// TwinCAT 3 PLC project MiseEnRoute
// libraries:
//   Maxon,1.0.0.0,Maxon Motor
//   Tc2_Standard,newest,Beckhoff Automation GmbH
//   Tc2_System,newest,Beckhoff Automation GmbH
//   Tc2_Utilities,newest,Beckhoff Automation GmbH
//   Tc3_Interfaces,3.3.0.0,Beckhoff Automation GmbH
//   Tc3_Module,3.3.6.0,Beckhoff Automation GmbH
// project tree:
//   / Blinking.TcTTO, GlobalImagePool.TcIPO (not stored), GlobalTextList.TcGTLO, Slow_Tasks.TcTTO, Standard.TcTTO, TestOperator.TcTTO, Visualization Manager.TcVMO (not stored)
//   Data types/ ETHERCAT.TcDUT, FLAGS.TcDUT, FLOWMETER_CONTROL.TcDUT, FLOWMETER_SENSOR.TcDUT, FLOWMETER_VALUES.TcDUT, GEN_PARAMS.TcDUT, HMI_DB_ADS.TcDUT, PANEL_KEYS.TcDUT, PANEL_LEDS.TcDUT, PMAX_DI.TcDUT, PMAX_DO.TcDUT, POW_DI.TcDUT, POW_DO.TcDUT, PRESSURE_SENSOR.TcDUT, PRINT_DI.TcDUT, PRINT_DO.TcDUT, PROG_STEPS.TcDUT, PUMP_PARAMS.TcDUT, PUMP_PARAMS_DB.TcDUT, Q_DI.TcDUT, Q_DO.TcDUT, SAFETY_IN.TcDUT, SAFETY_OUT.TcDUT, VAC_DI.TcDUT, VAC_DO.TcDUT
//   Global Variables/ Constant_Variables.TcGVL, Events_Variables.TcGVL, Flag_Variables.TcGVL, IOs_Variables.TcGVL, TwinCAT_Configuration.TcGVL, Variable_Configuration.TcGVL
//   POUs/ AIS.TcPOU, CHECK_VALVES_SENSORS.TcPOU, EVENTS.TcPOU, GEMMA.TcPOU, MAIN.TcPOU, Q1_MOTOR.TcPOU, Q2_MOTOR.TcPOU, SAFETY.TcPOU, testop.TcPOU, USB.TcPOU
//   POUs/Carriers/ CONVEYOR.TcPOU, JIG.TcPOU, JIG_2ND.TcPOU
//   POUs/EH/ EH_FLOMETER.TcPOU, EH_IEEE754_TO_REAL.TcPOU
//   POUs/Functions/ CONVERT_MASS_TO_FLOW.TcPOU
//   POUs/HMI/ LEDS.TcPOU
//   POUs/Stations/ PMAX.TcPOU, PRINT.TcPOU, Q1.TcPOU, Q2.TcPOU, VAC.TcPOU
//   POUs/Water/ WATER_TANK.TcPOU, WATER_TANKS.TcPOU
//   POUs/WIKA/ WIKA_GET_VALUES.TcPOU
//   Visualizations/ FLAGS.TcVIS, GEMMA.TcVIS, Motor.TcVIS, P_MAX.TcVIS, Q1.TcVIS, Q2.TcVIS, VAC.TcVIS

CONFIGURATION MiseEnRoute
    RESOURCE PLC ON TwinCAT3
        TASK Blinking(INTERVAL := T#450000us, PRIORITY := 23);
        TASK Slow_Tasks(INTERVAL := T#200000us, PRIORITY := 22);
        TASK Standard(INTERVAL := T#10ms, PRIORITY := 20);
        TASK TestOperator(INTERVAL := T#100000us, PRIORITY := 21);
        PROGRAM LEDS WITH Blinking : LEDS;
        PROGRAM USB WITH Slow_Tasks : USB;
        PROGRAM MAIN WITH Standard : MAIN;
        PROGRAM testop WITH TestOperator : testop;
    END_RESOURCE
END_CONFIGURATION

// ---- Data types/ETHERCAT.TcDUT
TYPE ETHERCAT :
STRUCT

	POW_COUPLER_STATUS:UINT;
	VAC_COUPLER_STATUS:UINT;
	Q1_COUPLER_STATUS:UINT;
	Q2_COUPLER_STATUS:UINT;
	PMAX_COUPLER_STATUS:UINT;
	PRINT_COUPLER_STATUS:UINT;

END_STRUCT
END_TYPE

// ---- Data types/FLAGS.TcDUT
TYPE FLAGS :
STRUCT

	INIT_OK:BOOL;
	INIT_CHECK_VALVES_SENSORS:BOOL;
	SAFETY_OK:BOOL;
	MANUAL:BOOL;
	AUTO:BOOL;
	VAC_STATUS: BOOL;
	JIG_VAC_STATUS: BOOL;
	Q1_STATUS: BOOL;
	Q2_STATUS: BOOL;
	PMAX_STATUS: BOOL;
	PRINT_STATUS: BOOL;
	JIG_Q1_STATUS: BOOL;
	JIG_Q2_STATUS: BOOL;
	JIG_PMAX_STATUS: BOOL;
	JIG_PRINT_STATUS: BOOL;
	VAC_RELEASE_CARRIER:BOOL;
	Q1_RELEASE_CARRIER:BOOL;
	Q2_RELEASE_CARRIER:BOOL;
	PMAX_RELEASE_CARRIER:BOOL;
	PRINT_RELEASE_CARRIER:BOOL;
	DOORS_OPEN:BOOL;
	F2_END:BOOL;
	GEMMA: STRING;
	MOTOR_Q1_INIT_OK:BOOL;
	MOTOR_Q1_POSITION:DINT;
	MOTOR_Q2_INIT_OK:BOOL;
	MOTOR_Q2_POSITION:DINT;



END_STRUCT
END_TYPE

// ---- Data types/FLOWMETER_CONTROL.TcDUT
TYPE FLOWMETER_CONTROL :
STRUCT

	SET_TOT: USINT;
	SET_MODE: USINT;

END_STRUCT
END_TYPE

// ---- Data types/FLOWMETER_SENSOR.TcDUT

(************************************************************************************************
*
*Variables structure for E&H flowmeter PROMAS 83A
*
***********************************************************************************************)


TYPE FLOWMETER_SENSOR :
STRUCT

	A1 :ARRAY[0..4] OF USINT;
	A2 :ARRAY[0..4] OF USINT;
	A3 :ARRAY[0..4] OF USINT;
	A4 :ARRAY[0..4] OF USINT;
	A5 :ARRAY[0..4] OF USINT;
	A6 :ARRAY[0..4] OF USINT;
	TOT :ARRAY[0..4] OF USINT;

END_STRUCT
END_TYPE

// ---- Data types/FLOWMETER_VALUES.TcDUT
TYPE FLOWMETER_VALUES :
STRUCT
	MassFlow:REAL;
	VolumeFlow:REAL;
	CorrectedVolueFLow:REAL;
	Density:REAL;
	ReferenceDensity:REAL;
	Temperature:REAL;
	TotalMass:REAL;
END_STRUCT
END_TYPE

// ---- Data types/GEN_PARAMS.TcDUT
TYPE GEN_PARAMS :
STRUCT

	USE_JIG_OP2:BOOL:=TRUE; (*Use or not the jig for the operator 2 - Right - *)

END_STRUCT
	END_TYPE

// ---- Data types/HMI_DB_ADS.TcDUT
TYPE HMI_DB_ADS :
STRUCT

	MANUAL				:REAL; (*Variables en provenance de la DB depuis le HMI*)
	AUTO				:REAL;
	NOT_AUS_RESET		:REAL;


END_STRUCT
END_TYPE

// ---- Data types/PANEL_KEYS.TcDUT
TYPE PANEL_KEYS :
STRUCT

	KEY1:BOOL;
	KEY2:BOOL;
	KEY3:BOOL;
	KEY4:BOOL;
	KEY5:BOOL;
	KEY6:BOOL;
	KEY7:BOOL;
	KEY8:BOOL;
	KEY9:BOOL;
	KEY10:BOOL;


END_STRUCT
END_TYPE

// ---- Data types/PANEL_LEDS.TcDUT
TYPE PANEL_LEDS :
STRUCT

	LED1:BOOL;
	LED2:BOOL;
	LED3:BOOL;
	LED4:BOOL;
	LED5:BOOL;
	LED6:BOOL;
	LED7:BOOL;
	LED8:BOOL;
	LED9:BOOL;
	LED10:BOOL;


END_STRUCT
END_TYPE

// ---- Data types/PMAX_DI.TcDUT
(************************************************************************************************
*
*Max pressure DI
*
***********************************************************************************************)

TYPE PMAX_DI :
STRUCT

	WAGON_WAITING:BOOL;
	WAGON_PRESENT:BOOL;
	WAGON_AWAY:BOOL;
	CYLINDER_TOP_IN:BOOL;
	CYLINDER_TOP_OUT:BOOL;
	CYLINDER_BOT_IN:BOOL;
	CYLINDER_BOT_OUT:BOOL;
	POWER_CYLINDER_IN:BOOL;
	POWER_CYLINDER_OUT:BOOL;
	Q3_OK:BOOL; 					(*Alim pompe*)
	WATER_TANK_HIGH:BOOL;
	WATER_TANK_LOW:BOOL;

END_STRUCT
END_TYPE

// ---- Data types/PMAX_DO.TcDUT
(************************************************************************************************
*
*Max pressure DO
*
***********************************************************************************************)

TYPE PMAX_DO :
STRUCT

	WAGON_WAIT_CYLINDER:BOOL;
	WAGON_LOCK_CYLINDER:BOOL;
	WAGON_STOP_CYLINDER:BOOL;
	HYDRO_CYLINDER_TOP:BOOL;
	HYDRO_CYLINDER_BOT:BOOL;
	ELECTR_CYLINDER:BOOL;
	Y7:BOOL;
	Y8:BOOL;
	PUMP_POWER:BOOL;
	PRESSURE_VALVE:BOOL;
	WATER_TANK_VALVE:BOOL;
	FLOW_STOP_VALVE:BOOL;
	FLOW_STOP_BOTT:BOOL;

END_STRUCT
END_TYPE

// ---- Data types/POW_DI.TcDUT

(************************************************************************************************
*
*Variables structure for the digitals intputs of the POWER module
*
***********************************************************************************************)


TYPE POW_DI :
STRUCT

	Q5_OK:BOOL; 		(* Disjoncteur Alimentation Chroma OK*)
	Q6_OK:BOOL;		(* Disjoncteur Alimentation Stations OK*)
	Q7_OK:BOOL;			(* Disjoncteur Moteurs L1L2L3 OK*)
	Q8_OK:BOOL;		(* Protection moteur 1 OK *)
	Q9_OK:BOOL;		(* Protection moteur 2 OK*)
	Q10_OK:BOOL;		(* Protection moteur 3 OK*)
	Q11_OK:BOOL;		(* Protection moteur 4 OK*)

END_STRUCT
END_TYPE

// ---- Data types/POW_DO.TcDUT

(************************************************************************************************
*
*Variables structure for the digitals ouputs of the POWER module
*
***********************************************************************************************)

TYPE POW_DO :
STRUCT

	HMI_LED_GREEN:BOOL;
	HMI_LED_ORANGE:BOOL;
	HMI_LED_RED:BOOL;
	HMI_LED_BLUE:BOOL;
	CONVEYOR_RELAIS:BOOL;


END_STRUCT
END_TYPE

// ---- Data types/PRESSURE_SENSOR.TcDUT

(************************************************************************************************
*
*Variables structure for WIKA pressure sensor
*
***********************************************************************************************)

TYPE PRESSURE_SENSOR :
STRUCT

	VALUE :ARRAY [0..7] OF USINT;

END_STRUCT
END_TYPE

// ---- Data types/PRINT_DI.TcDUT
(************************************************************************************************
*
*Printer DI
*
***********************************************************************************************)


TYPE PRINT_DI :
STRUCT

	WAGON_WAITING:BOOL;
	WAGON_PRESENT:BOOL;
	WAGON_AWAY:BOOL;
	Q3_OK:BOOL; 					(*Alim pompe*)
	WATER_TANK_HIGH:BOOL;
	WATER_TANK_LOW:BOOL;
	ASK_RELEASE_JIG_OP1:BOOL;
	ASK_RELEASE_JIG_OP2:BOOL;
	GRIPPER_OPEN:BOOL;
	GRIPPER_CLOSED:BOOL;
	X_IN:BOOL;
	X_OUT:BOOL;
	Z_UP:BOOL;
	Z_DOWN:BOOL;

END_STRUCT
END_TYPE

// ---- Data types/PRINT_DO.TcDUT
(************************************************************************************************
*
*Printer DO
*
***********************************************************************************************)

TYPE PRINT_DO :
STRUCT

	WAGON_WAIT_CYLINDER:BOOL;
	WAGON_LOCK_CYLINDER:BOOL;
	WAGON_STOP_CYLINDER:BOOL;
	EJECTION_CYLINDER_X:BOOL;
	EJECTION_CYLINDER_Z:BOOL;
	EJECTION_GRIPPER:BOOL;
	Y7:BOOL;
	Y8:BOOL;
	PUMP_POWER:BOOL;
	WATER_TANK_VALVE:BOOL;

END_STRUCT
END_TYPE

// ---- Data types/PROG_STEPS.TcDUT
TYPE PROG_STEPS :
STRUCT

	VAC_STEP:INT;
	Q1_STEP:INT;
	Q2_STEP:INT;
	PMAX_STEP:INT;
	PRINT_STEP:INT;


END_STRUCT
END_TYPE

// ---- Data types/PUMP_PARAMS.TcDUT
TYPE PUMP_PARAMS :
STRUCT

	VAC_ENABLE:BOOL					:=FALSE;				(*Enable Test*)
	VAC_PUMPING_TIME:TIME			:=T#5s; 			(*Pumping delay to prepare the pump for the suction test *)
	VAC_MEASUREMENT_TIME:TIME		:=T#5s; 			(*Measurement time for the sunction pressure *)
	VAC_PRESSURE_LIMIT:REAL			:=-0.7; 			(*Vacuum pressure Limit Higher than this parameter -> NO GOOD [bar]*)

	Q1_ENABLE:BOOL					:=TRUE;				(*Enable Test*)
	Q1_PUMPING_TIME:TIME			:=T#20s; 			(*Pumping delay to prepare the pump for the flow rate test *)
	Q1_MEASUREMENT_TIME:TIME		:=T#10s; 			(*Measurement time for the flow rate*)
	Q1_FLOW_TARGET:REAL				:=350; 				(*Flow rate target [ml/min]*)
	Q1_FLOW_LIMIT_UP:REAL			:=800; 				(*Flow rate Uper limit. Q>This limit -> NO GOOD [ml/min]*)
	Q1_FLOW_LIMIT_DOWN:REAL			:=100; 				(*Flow rate Lower limit. Q<This limit -> NO GOOD [ml/min]*)
	Q1_PRESSURE_TARGET:REAL			:=8; 				(*Pressure target [bar]*)
	Q1_PRESSURE_LIMIT_UP:REAL		:=15; 				(*Pressure Uper limit. p>This limit -> NO GOOD [bar]*)
	Q1_PRESSURE_LIMIT_DOWN:REAL		:=4;	 			(*Pressure Lower limit. p<This limit -> NO GOOD [bar]*)
	Q1_MAX_FLOW:BOOL				:=FALSE;			(*Use the max flow bypass*)

	Q2_ENABLE:BOOL					:=TRUE;				(*Enable Test*)
	Q2_PUMPING_TIME:TIME			:=T#20s; 			(*Pumping delay to prepare the pump for the flow rate test *)
	Q2_MEASUREMENT_TIME:TIME		:=T#10s; 			(*Measurement time for the flow rate*)
	Q2_FLOW_TARGET:REAL				:=350; 				(*Flow rate target [ml/min]*)
	Q2_FLOW_LIMIT_UP:REAL			:=800; 				(*Flow rate Uper limit. Q>This limit -> NO GOOD [ml/min]*)
	Q2_FLOW_LIMIT_DOWN:REAL			:=100; 				(*Flow rate Lower limit. Q<This limit -> NO GOOD [ml/min]*)
	Q2_PRESSURE_TARGET:REAL			:=8; 				(*Pressure target [bar]*)
	Q2_PRESSURE_LIMIT_UP:REAL		:=15; 				(*Pressure Uper limit. p>This limit -> NO GOOD [bar]*)
	Q2_PRESSURE_LIMIT_DOWN:REAL		:=4;	 			(*Pressure Lower limit. p<This limit -> NO GOOD [bar]*)
	Q2_MAX_FLOW:BOOL				:=FALSE;			(*Use the max flow bypass*)

	PMAX_ENABLE:BOOL				:=FALSE;				(*Enable Test*)
	PMAX_PUMPING_TIME:TIME			:=T#10s; 			(*Pumping delay to prepare the pump for the max pressure test *)
	PMAX_MEASUREMENT_TIME:TIME		:=T#8s; 			(*Measurement time for the max pressure test *)
	PMAX_PRESSURE_LIMIT:REAL		:=10; 				(*Max pressure lower than this parameter -> NO GOOD [bar]*)
	PMAX_PRESSURE_LOOSE_TIME:TIME	:=T#3s;				(*Valves Tightness test duration*)

	PRINT_ENABLE:BOOL				:=TRUE;			(*Enable Test*)

END_STRUCT
END_TYPE

// ---- Data types/PUMP_PARAMS_DB.TcDUT
TYPE PUMP_PARAMS_DB :
STRUCT


	VAC_ENABLE:REAL					;				(*Enable Test*)
	VAC_PUMPING_TIME:REAL			; 				(*Pumping delay to prepare the pump for the suction test *)
	VAC_MEASUREMENT_TIME:REAL		; 				(*Measurement time for the sunction pressure *)
	VAC_PRESSURE_LIMIT:REAL			; 				(*Vacuum pressure Limit Higher than this parameter -> NO GOOD [bar]*)

	Q1_ENABLE:REAL					;				(*Enable Test*)
	Q1_PUMPING_TIME:REAL				; 				(*Pumping delay to prepare the pump for the flow rate test *)
	Q1_MEASUREMENT_TIME:REAL		; 				(*Measurement time for the flow rate*)
	Q1_FLOW_TARGET:REAL				; 				(*Flow rate target [ml/min]*)
	Q1_FLOW_LIMIT_UP:REAL				; 				(*Flow rate Uper limit. Q>This limit -> NO GOOD [ml/min]*)
	Q1_FLOW_LIMIT_DOWN:REAL			; 				(*Flow rate Lower limit. Q<This limit -> NO GOOD [ml/min]*)
	Q1_PRESSURE_TARGET:REAL		; 				(*Pressure target [bar]*)
	Q1_PRESSURE_LIMIT_UP:REAL		; 				(*Pressure Uper limit. p>This limit -> NO GOOD [bar]*)
	Q1_PRESSURE_LIMIT_DOWN:REAL	;	 			(*Pressure Lower limit. p<This limit -> NO GOOD [bar]*)
	Q1_MAX_FLOW:REAL					;				(*Use the max flow bypass*)

	Q2_ENABLE:REAL					;				(*Enable Test*)
	Q2_PUMPING_TIME:REAL				; 				(*Pumping delay to prepare the pump for the flow rate test *)
	Q2_MEASUREMENT_TIME:REAL		; 				(*Measurement time for the flow rate*)
	Q2_FLOW_TARGET:REAL				; 				(*Flow rate target [ml/min]*)
	Q2_FLOW_LIMIT_UP:REAL				; 				(*Flow rate Uper limit. Q>This limit -> NO GOOD [ml/min]*)
	Q2_FLOW_LIMIT_DOWN:REAL			; 				(*Flow rate Lower limit. Q<This limit -> NO GOOD [ml/min]*)
	Q2_PRESSURE_TARGET:REAL		; 				(*Pressure target [bar]*)
	Q2_PRESSURE_LIMIT_UP:REAL		; 				(*Pressure Uper limit. p>This limit -> NO GOOD [bar]*)
	Q2_PRESSURE_LIMIT_DOWN:REAL	;	 			(*Pressure Lower limit. p<This limit -> NO GOOD [bar]*)
	Q2_MAX_FLOW:REAL					;				(*Use the max flow bypass*)

	PMAX_ENABLE:REAL					;				(*Enable Test*)
	PMAX_PUMPING_TIME:REAL			; 				(*Pumping delay to prepare the pump for the max pressure test *)
	PMAX_MEASUREMENT_TIME:REAL	; 				(*Measurement time for the max pressure test *)
	PMAX_PRESSURE_LIMIT:REAL		; 				(*Max pressure lower than this parameter -> NO GOOD [bar]*)

	PRINT_ENABLE:REAL				;				(*Enable Test*)


END_STRUCT
END_TYPE

// ---- Data types/Q_DI.TcDUT
(************************************************************************************************
*
*Flowmeter stations DI
*
***********************************************************************************************)

TYPE Q_DI :
STRUCT


	WAGON_WAITING:BOOL;
	WAGON_PRESENT:BOOL;
	WAGON_AWAY:BOOL;
	CYLINDER_TOP_IN:BOOL;
	CYLINDER_TOP_OUT:BOOL;
	CYLINDER_BOT_IN:BOOL;
	CYLINDER_BOT_OUT:BOOL;
	POWER_CYLINDER_IN:BOOL;
	POWER_CYLINDER_OUT:BOOL;
	Q3_OK:BOOL; 					(*Alim pompe*)
	WATER_TANK_HIGH:BOOL;
	WATER_TANK_LOW:BOOL;

END_STRUCT
END_TYPE

// ---- Data types/Q_DO.TcDUT
(************************************************************************************************
*
*Flowmeter stations DI
*
***********************************************************************************************)

TYPE Q_DO :
STRUCT


	WAGON_WAIT_CYLINDER:BOOL;
	WAGON_LOCK_CYLINDER:BOOL;
	WAGON_STOP_CYLINDER:BOOL;
	HYDRO_CYLINDER_TOP:BOOL;
	HYDRO_CYLINDER_BOT:BOOL;
	ELECTR_CYLINDER:BOOL;
	Y7:BOOL;
	Y8:BOOL;
	PUMP_POWER:BOOL;
	MAX_FLOW_VALVE:BOOL;
	WATER_TANK_VALVE:BOOL;
	FLOW_STOP_VALVE:BOOL;
	FLOW_STOP_BOTT:BOOL;

END_STRUCT
END_TYPE

// ---- Data types/SAFETY_IN.TcDUT
TYPE SAFETY_IN :
STRUCT

	DOORS_FBerr:BOOL;
	DOORS_COMerr:BOOL;
	DOORS_State:USINT;
	DOOR_VAC_CLOSED:BOOL;
	DOOR_Q1_CLOSED:BOOL;
	DOOR_Q2_CLOSED:BOOL;
	DOOR_PMAX_CLOSED:BOOL;
	DOOR_PRINT_CLOSED:BOOL;

	NOT_AUS_FBerr:BOOL;
	NOT_AUS_COMerr:BOOL;
	NOT_AUS_State:USINT;

END_STRUCT
END_TYPE

// ---- Data types/SAFETY_OUT.TcDUT
TYPE SAFETY_OUT :
STRUCT

	DOORS_RUN:BOOL;
	DOORS_ErrAck:BOOL;

	NOT_AUS_RUN:BOOL;
	NOT_AUS_ErrAck:BOOL;

	NOT_AUS_RESET:BOOL;

END_STRUCT
END_TYPE

// ---- Data types/VAC_DI.TcDUT
(************************************************************************************************
*
*Vacuum station DI
*
***********************************************************************************************)

TYPE VAC_DI :
STRUCT

	WAGON_WAITING:BOOL;
	WAGON_PRESENT:BOOL;
	WAGON_AWAY:BOOL;
	CYLINDER_TOP_IN:BOOL;
	CYLINDER_TOP_OUT:BOOL;
	CYLINDER_BOT_IN:BOOL;
	CYLINDER_BOT_OUT:BOOL;
	POWER_CYLINDER_IN:BOOL;
	POWER_CYLINDER_OUT:BOOL;
	Q3_OK:BOOL; 					(*Alim pompe*)
	WATER_TANK_HIGH:BOOL;
	WATER_TANK_LOW:BOOL;
	AIR_PRESSURE_OK:BOOL;


END_STRUCT
END_TYPE

// ---- Data types/VAC_DO.TcDUT
(************************************************************************************************
*
*Vacuum station DO
*
***********************************************************************************************)

TYPE VAC_DO :
STRUCT

	WAGON_WAIT_CYLINDER:BOOL;
	WAGON_LOCK_CYLINDER:BOOL;
	WAGON_STOP_CYLINDER:BOOL;
	HYDRO_CYLINDER_TOP:BOOL;
	HYDRO_CYLINDER_BOT:BOOL;
	ELECTR_CYLINDER:BOOL;
	WAGON_OPERATOR1:BOOL;
	WAGON_OPERATOR2:BOOL;
	PUMP_POWER:BOOL;
	VACUUM_VALVE:BOOL;
	WATER_TANK_VALVE:BOOL;
	AIR_VALVE:BOOL;
	FLOW_STOP_VALVE:BOOL;


END_STRUCT
END_TYPE

// ---- Global Variables/Constant_Variables.TcGVL
{attribute 'Tc2GvlVarNames'}
VAR_GLOBAL CONSTANT
	(********************
	*
	* Times
	*
	************************)

	CARRIER_RELEASE_DELAY						:TIME:= t#1s;			(*Delay between the release of the carrier on the main jig and the output of the CYLINDER_STOP*)
	CARRIER_STOP_DELAY							:TIME:= t#100ms;		(*Delay between the release of the carrier on the second jig and the output of the CYLINDER_WAIT*)
	PULSE_RELEASE_JIG_OP							:TIME:= t#250ms;		(*Duration of the pulse to release a carrier on the Operators jig*)
	DELAY_EJECT_CARRIERS						:TIME:= t#30s;			(*Time for release all the carriers present in the tunel during the initialisation *)
	TIMEOUT_WATER_TANK							:TIME:= t#500s;			(*Delay before an alarm during the fullfil of a watertank*)
	DRY_DELAY										:TIME:= T#1s;

	(********************
	*
	* Motor
	*
	************************)
	MOTOR_Q1_INITIAL_POS							:DINT:=10000;			(*Initial position of the motor*)
	MOTOR_Q1_POSITION_MAX						:DINT:=38000;		(*Butée soft du moteur*)
	MOTOR_Q2_INITIAL_POS							:DINT:=15000;			(*Initial position of the motor*)
	MOTOR_Q2_POSITION_MAX						:DINT:=36000;		(*Butée soft du moteur*)

END_VAR

VAR_GLOBAL

	(********************
	*
	* Config
	*
	************************)

	PUMP_PARAMS 									: PUMP_PARAMS;		(*Paramètre de test qu viennent depuis Labview*)

	GEN_PARAMS 									: GEN_PARAMS;


END_VAR

// ---- Global Variables/Events_Variables.TcGVL
{attribute 'Tc2GvlVarNames'}
VAR_GLOBAL


	(*EVENT PLC Started*)
	bSetEvent_1000_1 		:BOOL := FALSE; (*Set to lunch the event*)
	bQuitEvent_1000_1 		:BOOL := FALSE; (* Status of the confirmation *)
	LogEvent_1000_1 		:FB_SimpleAdsLogEvent; (* FB pour l'évenement *)

	(*EVENT Initializing*)
	bSetEvent_1000_2 		:BOOL := FALSE; (*Set to lunch the event*)
	bQuitEvent_1000_2 		:BOOL := FALSE; (* Status of the confirmation *)
	LogEvent_1000_2 		:FB_SimpleAdsLogEvent; (* FB pour l'évenement *)


END_VAR

// ---- Global Variables/Flag_Variables.TcGVL
{attribute 'Tc2GvlVarNames'}
VAR_GLOBAL


	FLAGS 				AT%M*: FLAGS;


	SAFETY_IN 			AT%I*: SAFETY_IN;
	SAFETY_OUT 			AT%Q*: SAFETY_OUT;

	ETHERCAT 			AT%I*:ETHERCAT;

	RUN_CG				:BOOL:=FALSE;
	CG_DELAY			:TIME:=T#15m;

(*
Status code for ETHERCAT coupler state

0x___1 = Slave in 'INIT' state
0x___2 = Slave in 'PREOP' state
0x___3 = Slave in 'BOOT' state
0x___4 = Slave in 'SAFEOP' state
0x___8 = Slave in 'OP' state
0x001_ = Slave signals error
0x002_ = Invalid vendorId, productCode... read
0x004_ = Initialization error occurred
0x008_ = Slave disabled
0x010_ = Slave not present
0x020_ = Slave signals link error
0x040_ = Slave signals missing link
0x080_ = Slave signals unexpected link
0x100_ = Communication port A
0x200_ = Communication port B
0x400_ = Communication port C
0x800_ = Communication port D

*)



END_VAR

// ---- Global Variables/IOs_Variables.TcGVL
{attribute 'Tc2GvlVarNames'}
VAR_GLOBAL


(************************************************************************************************
*
*General
*
***********************************************************************************************)
	PROG_STEPS:PROG_STEPS;

(************************************************************************************************
*
*Power Cabinet variables
*
***********************************************************************************************)

	POW_DI AT%IW100: POW_DI;
	POW_DO AT%QW100:POW_DO;

	KEY1 AT%I*:BOOL;
	LED1 AT%Q*:BOOL;

(************************************************************************************************
*
*Vacuum station variables
*
***********************************************************************************************)

	VAC_DI AT%IW200: VAC_DI;
	VAC_DO AT%QW200:VAC_DO;

	VAC_VACUUM_SENSOR AT%IW230: PRESSURE_SENSOR; (* Valeurs du capteur *)
	VAC_VACUMM_SENSOR_VALUE:REAL; (*Valeur réel*)

(************************************************************************************************
*
*Q1 station variables
*
***********************************************************************************************)

	Q1_DI AT%IW300: Q_DI;
	Q1_DO AT%QW300:Q_DO;

	Q1_PRESSURE_SENSOR AT%IW330: PRESSURE_SENSOR; (*Valeurs du capteur*)
	Q1_PRESSURE_SENSOR_VALUE:REAL;(*Valeur réel*)
	Q1_CALCULETED_FLOW:REAL ;

	Q1_FLOWMETER AT%IW340:FLOWMETER_SENSOR; (*Valeurs du capteur*)
	Q1_FLOWMETER_VALUES :FLOWMETER_VALUES;(*Valeurs réels*)
	Q1_FLOWMETER_CONTROL AT%QW350:FLOWMETER_CONTROL;(*Variables de commande du débitmètre*)

	Q1_CURRENT:REAL;

(************************************************************************************************
*
*Q2 station variables
*
***********************************************************************************************)

	Q2_DI AT%IW400: Q_DI;
	Q2_DO AT%QW400:Q_DO;

	Q2_PRESSURE_SENSOR AT%IW430: PRESSURE_SENSOR;
	Q2_PRESSURE_SENSOR_VALUE:REAL;
	Q2_CALCULETED_FLOW:REAL ;

	Q2_FLOWMETER AT%IW440:FLOWMETER_SENSOR;
	Q2_FLOWMETER_VALUES :FLOWMETER_VALUES;
	Q2_FLOWMETER_CONTROL AT%QW450:FLOWMETER_CONTROL;(*Variables de commande du débitmètre*)

	Q2_CURRENT:REAL;

(************************************************************************************************
*
*PMAX station variables
*
***********************************************************************************************)

	PMAX_DI AT%IW500: PMAX_DI;
	PMAX_DO AT%QW500: PMAX_DO;

	PMAX_PRESSURE_SENSOR AT%IW530: PRESSURE_SENSOR;
	PMAX_PRESSURE_SENSOR_VALUE:REAL;

	PMAX_PRESSURE_LOOSE:REAL;

(************************************************************************************************
*
*PRINT station variables
*
***********************************************************************************************)

	PRINT_DI AT%IW600: PRINT_DI;
	PRINT_DO AT%QW600: PRINT_DO;

	PRINT_PUMP_STATUS	:BOOL; (*0-> pompe mauvaise / 1-> pompe bonne*)

	CAN_OPEN_Q1_DIAGAT AT%I*:BOOL;

	CAN_OPEN_Q2_DIAGAT AT%I*:BOOL;

(************************************************************************************************
*
*Current measurement
*
***********************************************************************************************)
	Q1_Multimeter_mode	AT%Q*:SINT := 3;
	Q2_Multimeter_mode	AT%Q*:SINT := 3;
(*
0 0x00 DC voltage
1 0x01 AC voltage
2 0x02 DC current
3 0x03 AC current
*)

	Q1_Multimeter_range AT%Q* :SINT := 1;
	Q2_Multimeter_range AT%Q* :SINT := 1;

(*
255 0xFF 300 mV / 100 mA
0 0x00  3 V / 1 A 
1 0x01 30 V / 10 A 
2 0x02 300 V (voltage only)  
*)

	Q1_Multimeter_value AT%I*:DINT;
	Q2_Multimeter_value AT%I*:DINT;


END_VAR

// ---- Global Variables/TwinCAT_Configuration.TcGVL
{attribute 'Tc2GvlVarNames'}
(* Generated automatically by TwinCAT - (read only) *)
VAR_CONFIG
	.SAFETY_IN AT %IB1528 : SAFETY_IN;
	.SAFETY_OUT AT %QB612 : SAFETY_OUT;
	.ETHERCAT AT %IB1512 : ETHERCAT;
	.KEY1 AT %IX1552.0 : BOOL;	(*  ~ {LinkedWith:TIID^Device 1 (USB)^Box 0 (CPX8XX)^Term 1 (CPx9xx-12)^Channel 1^Key 1} *)
	.LED1 AT %QX624.0 : BOOL;	(*  ~ {LinkedWith:TIID^Device 1 (USB)^Box 0 (CPX8XX)^Term 1 (CPx9xx-12)^Channel 1^LED 1} *)
	.CAN_OPEN_Q1_DIAGAT AT %IX1524.0 : BOOL;	(*  ~ {LinkedWith:TIID^CanOPEN Q1 (EL6751)^Entrées^DiagFlag} *)
	.CAN_OPEN_Q2_DIAGAT AT %IX1540.0 : BOOL;	(*  ~ {LinkedWith:TIID^CanOPEN Q2 (EL6751)^Entrées^DiagFlag} *)
	.Q1_Multimeter_mode AT %QB620 : SINT;	(*  ~ {LinkedWith:TIID^I/O (Ethercat)^Q1 (EK1101)^Terme 41 (EL3681)^SAI Range^Mode} *)
	.Q2_Multimeter_mode AT %QB621 : SINT;	(*  ~ {LinkedWith:TIID^I/O (Ethercat)^Q2 (EK1101)^Terme 114 (EL3681)^SAI Range^Control^Mode} *)
	.Q1_Multimeter_range AT %QB622 : SINT;	(*  ~ {LinkedWith:TIID^I/O (Ethercat)^Q1 (EK1101)^Terme 41 (EL3681)^SAI Range^Range} *)
	.Q2_Multimeter_range AT %QB623 : SINT;	(*  ~ {LinkedWith:TIID^I/O (Ethercat)^Q2 (EK1101)^Terme 114 (EL3681)^SAI Range^Control^Range} *)
	.Q1_Multimeter_value AT %IB1544 : DINT;	(*  ~ {LinkedWith:TIID^I/O (Ethercat)^Q1 (EK1101)^Terme 41 (EL3681)^SAI Inputs^Value} *)
	.Q2_Multimeter_value AT %IB1548 : DINT;	(*  ~ {LinkedWith:TIID^I/O (Ethercat)^Q2 (EK1101)^Terme 114 (EL3681)^SAI Inputs^Value} *)
END_VAR

// ---- Global Variables/Variable_Configuration.TcGVL
{attribute 'Tc2GvlVarNames'}
VAR_CONFIG
END_VAR

// ---- POUs/HMI/LEDS.TcPOU
PROGRAM LEDS
VAR
	M1_FB_GetPositionIs: FB_GetPositionIs;
	M1_FB_GetEnableState: FB_GetEnableState;

	M2_FB_GetPositionIs: FB_GetPositionIs;
	M2_FB_GetEnableState: FB_GetEnableState;
END_VAR

(****************************************************************************************************
*
* Gestion des lumières sur l'armoire de commande 
*
****************************************************************************************************)

IF GEMMA.STEP='D1' THEN
	POW_DO.HMI_LED_BLUE:=FALSE;
	POW_DO.HMI_LED_RED:=TRUE;
	POW_DO.HMI_LED_ORANGE:=FALSE;
	POW_DO.HMI_LED_GREEN:=FALSE;
ELSIF GEMMA.STEP='A6' THEN
	POW_DO.HMI_LED_BLUE:=FALSE;
	POW_DO.HMI_LED_RED:=FALSE;
	POW_DO.HMI_LED_ORANGE:=TRUE;
	POW_DO.HMI_LED_GREEN:=FALSE;
ELSIF GEMMA.STEP='A1' THEN
	POW_DO.HMI_LED_BLUE:= NOT POW_DO.HMI_LED_BLUE;
	POW_DO.HMI_LED_RED:=FALSE;
	POW_DO.HMI_LED_ORANGE:=FALSE;
	POW_DO.HMI_LED_GREEN:=FALSE;
ELSIF GEMMA.STEP='F1' THEN
	POW_DO.HMI_LED_BLUE:=FALSE;
	POW_DO.HMI_LED_RED:=FALSE;
	POW_DO.HMI_LED_ORANGE:=FALSE;
	POW_DO.HMI_LED_GREEN:=TRUE;
ELSIF GEMMA.STEP='F4' THEN
	POW_DO.HMI_LED_BLUE:=FALSE;
	POW_DO.HMI_LED_RED:=FALSE;
	POW_DO.HMI_LED_ORANGE:=TRUE;
	POW_DO.HMI_LED_GREEN:=TRUE;
ELSE
    	POW_DO.HMI_LED_BLUE:=FALSE;
	POW_DO.HMI_LED_RED:=FALSE;
	POW_DO.HMI_LED_ORANGE:=FALSE;
	POW_DO.HMI_LED_GREEN:=FALSE;
END_IF;

(*INFO Moteur*)
M1_FB_GetPositionIs(
	ADSNetId:= '10.0.0.31.6.1',
	NodeId:= 1,
	Read:= TRUE
	);

M1_FB_GetEnableState(
	ADSNetId:= '10.0.0.31.6.1',
	NodeId:= 1,
	Read:= TRUE);


M2_FB_GetPositionIs(
	ADSNetId:= '10.0.0.31.8.1',
	NodeId:= 1,
	Read:= TRUE
	);

M2_FB_GetEnableState(
	ADSNetId:= '10.0.0.31.8.1',
	NodeId:= 1,
	Read:= TRUE);

END_PROGRAM

// ---- POUs/GEMMA.TcPOU
PROGRAM GEMMA
VAR
	STEP_A6: INT := 0;
	DELAY_EJECTION_CARRIERS: TON;
	EJECT_CARRIERS: BOOL;
	F2_END: BOOL;
	STEP: STRING(20);
END_VAR

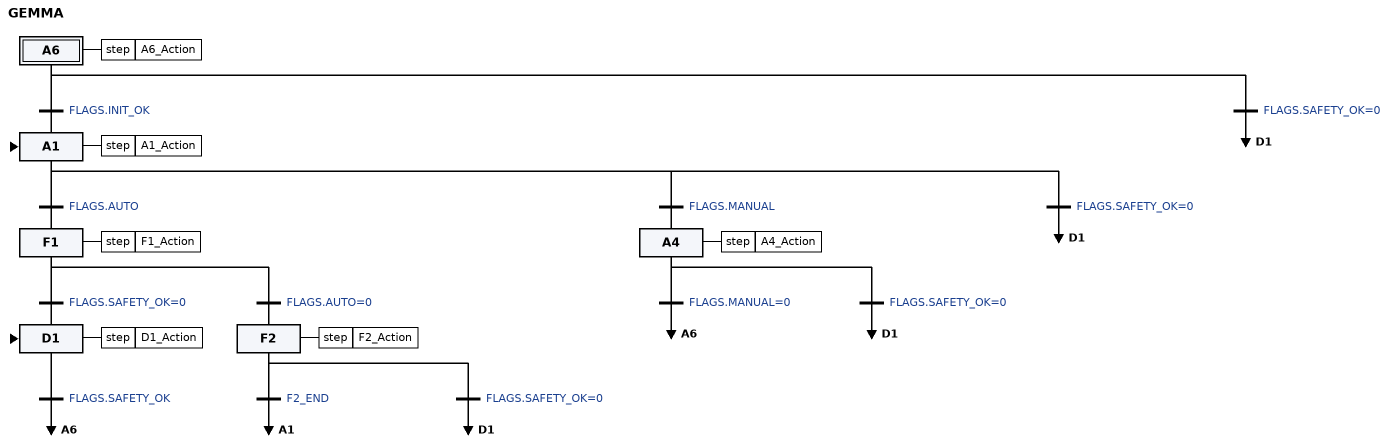
INITIAL_STEP A6_:  // name as stored: A6 
    A6_Action(N);  // step action
END_STEP
TRANSITION FROM A6_ TO A1
    := FLAGS.INIT_OK;
END_TRANSITION
TRANSITION FROM A6_ TO D1
    := FLAGS.SAFETY_OK=0;
END_TRANSITION
STEP A1:
    A1_Action(N);  // step action
END_STEP
TRANSITION FROM A1 TO F1
    := FLAGS.AUTO;
END_TRANSITION
TRANSITION FROM A1 TO A4
    := FLAGS.MANUAL;
END_TRANSITION
STEP A4:
    A4_Action(N);  // step action
END_STEP
TRANSITION FROM A4 TO A6
    := FLAGS.MANUAL=0;
END_TRANSITION
TRANSITION FROM A4 TO D1
    := FLAGS.SAFETY_OK=0;
END_TRANSITION
TRANSITION FROM A1 TO D1
    := FLAGS.SAFETY_OK=0;
END_TRANSITION
STEP F1:
    F1_Action(N);  // step action
END_STEP
TRANSITION FROM F1 TO D1
    := FLAGS.SAFETY_OK=0;
END_TRANSITION
TRANSITION FROM F1 TO F2
    := FLAGS.AUTO=0;
END_TRANSITION
STEP F2:
    F2_Action(N);  // step action
END_STEP
TRANSITION FROM F2 TO A1
    := F2_END;
END_TRANSITION
TRANSITION FROM F2 TO D1
    := FLAGS.SAFETY_OK=0;
END_TRANSITION
STEP D1:
    D1_Action(N);  // step action
END_STEP
TRANSITION FROM D1 TO A6
    := FLAGS.SAFETY_OK;
END_TRANSITION

ACTION A6_Action:
(**************************************************************
*
*
* Initialisation
*
*
***************************************************************)
STEP:='A6';

PMAX();
VAC();
Q1();
Q2();
(*CONVEYOR();*)


CASE STEP_A6 OF

0: (*Init*)
	STEP_A6:=STEP_A6+1;

1: (*Initialise valves and variables*)

	FLAGS.INIT_OK:=FALSE;
	FLAGS.INIT_CHECK_VALVES_SENSORS:=TRUE;

	FLAGS.VAC_RELEASE_CARRIER:=FALSE;
	FLAGS.Q1_RELEASE_CARRIER:=FALSE;
	FLAGS.Q2_RELEASE_CARRIER:=FALSE;
	FLAGS.PMAX_RELEASE_CARRIER:=FALSE;
	FLAGS.PRINT_RELEASE_CARRIER:=FALSE;

	FLAGS.MOTOR_Q1_INIT_OK:=FALSE;
	FLAGS.MOTOR_Q1_POSITION:=MOTOR_Q1_INITIAL_POS;

	VAC_DO.AIR_VALVE := FALSE;

	VAC_DO.ELECTR_CYLINDER := FALSE;
	VAC_DO.HYDRO_CYLINDER_BOT := FALSE;
	VAC_DO.HYDRO_CYLINDER_TOP := FALSE;

	VAC_DO.WAGON_LOCK_CYLINDER := FALSE;
	VAC_DO.WAGON_STOP_CYLINDER := FALSE;
	VAC_DO.WAGON_WAIT_CYLINDER := FALSE;

	VAC_DO.FLOW_STOP_VALVE := FALSE;
	VAC_DO.WATER_TANK_VALVE := FALSE;
	VAC_DO.PUMP_POWER := FALSE;
	VAC_DO.VACUUM_VALVE := FALSE;
	VAC_DO.WAGON_OPERATOR1:=TRUE;
	VAC_DO.WAGON_OPERATOR2:=TRUE;


	Q1_DO.ELECTR_CYLINDER := FALSE;
	Q1_DO.HYDRO_CYLINDER_BOT := FALSE;
	Q1_DO.HYDRO_CYLINDER_TOP := FALSE;
	Q1_DO.WAGON_LOCK_CYLINDER := FALSE;
	Q1_DO.WAGON_STOP_CYLINDER := FALSE;
	Q1_DO.WAGON_WAIT_CYLINDER := FALSE;
	Q1_DO.PUMP_POWER:=FALSE;
	Q1_DO.FLOW_STOP_BOTT:=FALSE;

	Q2_DO.ELECTR_CYLINDER := FALSE;
	Q2_DO.HYDRO_CYLINDER_BOT := FALSE;
	Q2_DO.HYDRO_CYLINDER_TOP := FALSE;
	Q2_DO.WAGON_LOCK_CYLINDER := FALSE;
	Q2_DO.WAGON_STOP_CYLINDER := FALSE;
	Q2_DO.WAGON_WAIT_CYLINDER := FALSE;
	Q2_DO.PUMP_POWER:=FALSE;
	Q2_DO.FLOW_STOP_BOTT:=TRUE;

	PMAX_DO.ELECTR_CYLINDER := FALSE;
	PMAX_DO.HYDRO_CYLINDER_BOT := FALSE;
	PMAX_DO.HYDRO_CYLINDER_TOP := FALSE;
	PMAX_DO.WAGON_LOCK_CYLINDER := FALSE;
	PMAX_DO.WAGON_STOP_CYLINDER := FALSE;
	PMAX_DO.WAGON_WAIT_CYLINDER := FALSE;
	PMAX_DO.PUMP_POWER:=FALSE;
	PMAX_DO.FLOW_STOP_BOTT:=FALSE;

	PRINT_DO.WAGON_LOCK_CYLINDER := FALSE;
	PRINT_DO.WAGON_STOP_CYLINDER := FALSE;
	PRINT_DO.WAGON_WAIT_CYLINDER := FALSE;


	STEP_A6:=STEP_A6+1;

2: (*Start AIR and wait for ejection of all carriers on the conveyor*)

	VAC_DO.AIR_VALVE := TRUE;
	POW_DO.CONVEYOR_RELAIS := TRUE;
	EJECT_CARRIERS:=TRUE;

	STEP_A6:=STEP_A6+1;

3: (* Wait carriers ejection *)

	IF DELAY_EJECTION_CARRIERS.Q THEN
		EJECT_CARRIERS:=FALSE;
		STEP_A6:=STEP_A6+1;
	END_IF;

4:(*Check valves sensors A IMPLEMENTER PLUS TARD *)
	IF FLAGS.INIT_CHECK_VALVES_SENSORS THEN
		;(*CHECK_VALVES_SENSORS();*)
		STEP_A6:=STEP_A6+1;
	ELSE
		STEP_A6:=STEP_A6+1;
	END_IF;

5: (*End of init *)

	FLAGS.INIT_OK:=TRUE;


ELSE
    ;
END_CASE;

(* FBs *)
DELAY_EJECTION_CARRIERS(IN:=EJECT_CARRIERS , PT:= DELAY_EJECT_CARRIERS);
END_ACTION

ACTION F2_Action:
STEP := 'F2';

VAC();
CONVEYOR();

IF VAC.STEP=10 THEN

F2_END:=TRUE;

END_IF;
END_ACTION

ACTION A1_Action:
(***************************************************************************
*
* A1
*
****************************************************************************)
STEP := 'A1';

F2_END:=FALSE;
END_ACTION

ACTION F1_Action:
(*********************************************************
*
* F1
*
************************************************************)

STEP := 'F1';

(* Station VAC *)
IF PUMP_PARAMS.VAC_ENABLE THEN
	VAC();
ELSE
	FLAGS.VAC_RELEASE_CARRIER:=TRUE;
END_IF;

(* Station Q1 *)
IF PUMP_PARAMS.Q1_ENABLE THEN
	Q1();
ELSE
	FLAGS.Q1_RELEASE_CARRIER:=TRUE;
END_IF;

(* Station Q2 *)
IF PUMP_PARAMS.Q2_ENABLE THEN
	Q2();
ELSE
	FLAGS.Q2_RELEASE_CARRIER:=TRUE;
END_IF;

(* Station PMAX *)
IF PUMP_PARAMS.PMAX_ENABLE THEN
	PMAX();
ELSE
	FLAGS.PMAX_RELEASE_CARRIER:=TRUE;
END_IF;

(* Station PRINT *)
IF PUMP_PARAMS.PRINT_ENABLE THEN
	PRINT();
ELSE
	FLAGS.PRINT_RELEASE_CARRIER:=TRUE;
END_IF;



CONVEYOR();
END_ACTION

ACTION A4_Action:
STEP:= 'A4';
END_ACTION

ACTION D1_Action:
(*****************************************************************
*
* NOT AUS state
*
******************************************************************)

	STEP := 'D1';

	FLAGS.INIT_OK:=FALSE;
	FLAGS.MOTOR_Q1_INIT_OK:=FALSE;
	FLAGS.AUTO:=FALSE;
	FLAGS.MANUAL:=FALSE;


	VAC_DO.AIR_VALVE := FALSE;
	POW_DO.CONVEYOR_RELAIS:=FALSE;

	VAC_DO.ELECTR_CYLINDER := FALSE;
	VAC_DO.HYDRO_CYLINDER_BOT := FALSE;
	VAC_DO.HYDRO_CYLINDER_TOP := FALSE;
	VAC_DO.WAGON_LOCK_CYLINDER := FALSE;
	VAC_DO.WAGON_STOP_CYLINDER := FALSE;
	VAC_DO.WAGON_WAIT_CYLINDER := FALSE;
	VAC_DO.PUMP_POWER:=FALSE;
	VAC_DO.WAGON_OPERATOR1:=TRUE;
	VAC_DO.WAGON_OPERATOR2:=FALSE;

	Q1_DO.ELECTR_CYLINDER := FALSE;
	Q1_DO.HYDRO_CYLINDER_BOT := FALSE;
	Q1_DO.HYDRO_CYLINDER_TOP := FALSE;
	Q1_DO.WAGON_LOCK_CYLINDER := FALSE;
	Q1_DO.WAGON_STOP_CYLINDER := FALSE;
	Q1_DO.WAGON_WAIT_CYLINDER := FALSE;
	Q1_DO.PUMP_POWER:=FALSE;

	Q2_DO.ELECTR_CYLINDER := FALSE;
	Q2_DO.HYDRO_CYLINDER_BOT := FALSE;
	Q2_DO.HYDRO_CYLINDER_TOP := FALSE;
	Q2_DO.WAGON_LOCK_CYLINDER := FALSE;
	Q2_DO.WAGON_STOP_CYLINDER := FALSE;
	Q2_DO.WAGON_WAIT_CYLINDER := FALSE;
	Q2_DO.PUMP_POWER:=FALSE;

	PMAX_DO.ELECTR_CYLINDER := FALSE;
	PMAX_DO.HYDRO_CYLINDER_BOT := FALSE;
	PMAX_DO.HYDRO_CYLINDER_TOP := FALSE;
	PMAX_DO.WAGON_LOCK_CYLINDER := FALSE;
	PMAX_DO.WAGON_STOP_CYLINDER := FALSE;
	PMAX_DO.WAGON_WAIT_CYLINDER := FALSE;
	PMAX_DO.PUMP_POWER:=FALSE;


	PRINT_DO.WAGON_LOCK_CYLINDER	:= FALSE;
	PRINT_DO.WAGON_STOP_CYLINDER 	:= FALSE;
	PRINT_DO.WAGON_WAIT_CYLINDER	:= FALSE;
	PRINT_DO.EJECTION_CYLINDER_X	:=FALSE;
	PRINT_DO.EJECTION_CYLINDER_Z	:=FALSE;
	PRINT_DO.EJECTION_GRIPPER		:=FALSE;

	STEP_A6:=0;


	CONVEYOR();
END_ACTION

END_PROGRAM

// ---- POUs/Stations/PMAX.TcPOU
PROGRAM PMAX
VAR
	STEP: INT := 0;
	R_TRIG1:R_TRIG;
	Presure_Delay: TON;
	FlowStop_Delay: TON;
	Start_FlowStop_Delay: BOOL;
	Pump_Delay: TON;
	Start_Pump_Delay: BOOL;
	Start_Presure_Delay: BOOL;
	Start_Tightness_Delay: BOOL;
	Tightness_Delay: TON;
	Tightness_1: REAL;
END_VAR

(*******************************************************
*
* Program fro the PMAX Test station
*
*
*********************************************************)
IF GEMMA.STEP='A6' THEN
	STEP:=0;
END_IF;


CASE STEP OF

0: (*Init*)
	Start_Pump_Delay:=FALSE;
	Start_Presure_Delay:=FALSE;
	Start_FlowStop_Delay:=FALSE;
	FLAGS.PMAX_STATUS:=0;
	FLAGS.PMAX_RELEASE_CARRIER:=0;
	STEP := STEP+10;

10: (*Wait main JIG Ready*)
	IF R_TRIG1.Q AND GEMMA.STEP='F1'  THEN
		FLAGS.PMAX_STATUS:=1;
		STEP := STEP+10;

	END_IF;

20: (*Continue if doors closed**************************************************************************)
	IF FLAGS.DOORS_OPEN=0 THEN
		STEP := STEP+10;
	END_IF;

30: (* Check hydraulique connexion OK*)
	PMAX_DO.HYDRO_CYLINDER_BOT:=TRUE;
	PMAX_DO.HYDRO_CYLINDER_TOP:=TRUE;
	PMAX_PRESSURE_LOOSE := 0;

	STEP := STEP+10;

40: (*Continue if doors closed**************************************************************************)
	IF FLAGS.DOORS_OPEN=0 THEN
		STEP := STEP+10;
	END_IF;

50: (* Wait hydraulique connexion OK*)
	IF PMAX_DI.CYLINDER_BOT_OUT AND PMAX_DI.CYLINDER_TOP_OUT THEN
		STEP := STEP+10;
	END_IF;

60: (*Continue if doors closed**************************************************************************)
	IF FLAGS.DOORS_OPEN=0 THEN
		STEP := STEP+10;
	END_IF;

70: (*Close electrical connexion *)
	PMAX_DO.ELECTR_CYLINDER:=TRUE;
	STEP := STEP+10;

80: (*Continue if doors closed**************************************************************************)
	IF FLAGS.DOORS_OPEN=0 THEN
		STEP := STEP+10;
	END_IF;

90:(*Wait electrical connexion closed*)
	IF PMAX_DI.POWER_CYLINDER_OUT THEN
		Start_Pump_Delay:=TRUE;
		PMAX_DO.PUMP_POWER:=TRUE;
		PMAX_DO.PRESSURE_VALVE:=FALSE;
		PMAX_DO.FLOW_STOP_BOTT:=TRUE;
		STEP := STEP+10;
	END_IF;

100: (*Continue if doors closed**************************************************************************)
	IF FLAGS.DOORS_OPEN=0 THEN
		STEP := STEP+10;
	END_IF;

110: (*Pump until end of delay*)
	IF Pump_Delay.Q THEN
		Start_Pump_Delay:=FALSE;
		PMAX_DO.PRESSURE_VALVE:=TRUE;
		Start_Presure_Delay:=TRUE;
		STEP := STEP+10;
	END_IF;

120: (*Continue if doors closed**************************************************************************)
	IF FLAGS.DOORS_OPEN=0 THEN
		STEP := STEP+10;
	END_IF;


130: (*Presure until end of delay*)
	IF Presure_Delay.Q THEN
		PMAX_DO.HYDRO_CYLINDER_BOT:=FALSE;
		Start_Presure_Delay:=FALSE;
		STEP := STEP+10;
	END_IF;

140: (*Continue if doors closed**************************************************************************)
	IF FLAGS.DOORS_OPEN=0 THEN
		STEP := STEP+10;
	END_IF;

150: (*Stop pump for valve tightness*)
		PMAX_DO.PUMP_POWER:=FALSE;
		Start_Tightness_Delay:=TRUE;
		Tightness_1:=PMAX_PRESSURE_SENSOR_VALUE;
		STEP := STEP+10;

160: (*Wait valve tightness test time*)
	IF Tightness_Delay.Q THEN
		PMAX_DO.PRESSURE_VALVE:=FALSE;
		PMAX_DO.FLOW_STOP_BOTT:=TRUE;
		PMAX_DO.PUMP_POWER:=TRUE;
		Start_Tightness_Delay:=FALSE;
		Start_FlowStop_Delay:=TRUE;
		PMAX_PRESSURE_LOOSE:=Tightness_1-PMAX_PRESSURE_SENSOR_VALUE;
		STEP := STEP+10;
	END_IF;


(***MODIFICATION POUR PRESSURE LOOSE TIGHTNESS AVANT CETTE LIGNE *************)
170: (*Delay before FLOWSTOP*)
	IF FlowStop_Delay.Q THEN
		PMAX_DO.FLOW_STOP_BOTT:=FALSE;
		PMAX_DO.PRESSURE_VALVE:=TRUE;
		PMAX_DO.PUMP_POWER:=FALSE;
		Start_FlowStop_Delay:=FALSE;
		STEP := STEP+10;
	END_IF;


180: (*Continue if doors closed**************************************************************************)
	IF FLAGS.DOORS_OPEN=0 THEN
		STEP := STEP+10;
	END_IF;


190: (*Release electrical and hydraulic connexion*)


	PMAX_DO.HYDRO_CYLINDER_TOP:=FALSE;
	PMAX_DO.ELECTR_CYLINDER:=FALSE;

	STEP := STEP+10;

200: (*Continue if doors closed**************************************************************************)
	IF FLAGS.DOORS_OPEN=0 THEN
		STEP := STEP+10;
	END_IF;

210:(*Wait all cylinders IN*)
	IF PMAX_DI.POWER_CYLINDER_IN AND PMAX_DI.CYLINDER_BOT_IN AND PMAX_DI.CYLINDER_TOP_IN THEN
		STEP := STEP+10;
	END_IF;

220: (*Continue if doors closed**************************************************************************)
	IF FLAGS.DOORS_OPEN=0 THEN
		STEP := STEP+10;
	END_IF;

230: (*Release carrier*)
	FLAGS.PMAX_RELEASE_CARRIER:=TRUE;
	STEP:=STEP+10;

240: (*Continue if doors closed**************************************************************************)
	IF FLAGS.DOORS_OPEN=0 THEN
		STEP := STEP+10;
	END_IF;

250: (*Wait carrier away*)
	IF PMAX_DI.WAGON_AWAY THEN
		STEP := 0;
	END_IF;



ELSE
    ;
END_CASE;

PROG_STEPS.PMAX_STEP:=STEP;

(*FBs*)
Pump_Delay(IN:= Start_Pump_Delay, PT:= PUMP_PARAMS.PMAX_PUMPING_TIME);
Presure_Delay(IN:= Start_Presure_Delay, PT:= PUMP_PARAMS.PMAX_MEASUREMENT_TIME);
FlowStop_Delay(IN:= Start_FlowStop_Delay, PT:= DRY_DELAY);
Tightness_Delay(IN:= Start_Tightness_Delay, PT:= PUMP_PARAMS.PMAX_PRESSURE_LOOSE_TIME);

R_TRIG1(CLK:= CONVEYOR.JIG_PMAX.STATUS);

END_PROGRAM

// ---- POUs/Carriers/CONVEYOR.TcPOU
PROGRAM CONVEYOR

VAR
	JIG_VAC: JIG;
	JIG_Q1:JIG;
	JIG_Q2: JIG;
	JIG_PMAX: JIG;
	JIG_PRINT: JIG;

	JIG_VAC_2nd: JIG_2ND;
	JIG_Q1_2nd: JIG_2ND;
	JIG_Q2_2nd: JIG_2ND;
	JIG_PMAX_2nd: JIG_2ND;
	JIG_PRINT_2nd: JIG_2ND;

	F_TRIG1:F_TRIG;
	PULSE_RELEASE_JIG_OP1:TP;
	PULSE_RELEASE_JIG_OP2: TP;

END_VAR
VAR_INPUT
END_VAR

(**********************************
*
* Gestion des posages Opérateur 1 et 2
*
********************************************)
IF (GEMMA.STEP='F1' OR GEMMA.STEP='F4') AND NOT(RUN_CG) THEN

	PULSE_RELEASE_JIG_OP1(IN:=PRINT_DI.ASK_RELEASE_JIG_OP1 , PT:= PULSE_RELEASE_JIG_OP );
	PULSE_RELEASE_JIG_OP2(IN:=PRINT_DI.ASK_RELEASE_JIG_OP2 , PT:= PULSE_RELEASE_JIG_OP );

	VAC_DO.WAGON_OPERATOR1:= NOT PULSE_RELEASE_JIG_OP1.Q;

	IF GEN_PARAMS.USE_JIG_OP2 THEN
		VAC_DO.WAGON_OPERATOR2:= NOT PULSE_RELEASE_JIG_OP2.Q;
	ELSE
		VAC_DO.WAGON_OPERATOR2:=FALSE;
	END_IF;


END_IF;

(*test*)
(*IF GEMMA.STEP='F1' OR GEMMA.STEP='F4' THEN
VAC_DO.WAGON_OPERATOR1:=FALSE;
VAC_DO.WAGON_OPERATOR2:=FALSE;
END_IF;*)
(*test*)

(**********************************
*
* Gestion des posages principaux
*
********************************************)
JIG_VAC(
	CARRIER_PRESENT:=VAC_DI.WAGON_PRESENT ,
	RELEASE_CARRIER:= FLAGS.VAC_RELEASE_CARRIER,
	STATUS=> FLAGS.JIG_VAC_STATUS,
	NEXT_JIG_STATUS:=Q1_DI.WAGON_WAITING,
	CYLINDER_STOP=> VAC_DO.WAGON_STOP_CYLINDER,
	CYLINDER_LOCK=> VAC_DO.WAGON_LOCK_CYLINDER);

JIG_Q1(
	CARRIER_PRESENT:=Q1_DI.WAGON_PRESENT ,
	RELEASE_CARRIER:= FLAGS.Q1_RELEASE_CARRIER,
	STATUS=> FLAGS.JIG_Q1_STATUS,
	NEXT_JIG_STATUS:=Q2_DI.WAGON_WAITING,
	CYLINDER_STOP=> Q1_DO.WAGON_STOP_CYLINDER,
	CYLINDER_LOCK=> Q1_DO.WAGON_LOCK_CYLINDER);

JIG_Q2(
	CARRIER_PRESENT:=Q2_DI.WAGON_PRESENT ,
	RELEASE_CARRIER:= FLAGS.Q2_RELEASE_CARRIER,
	STATUS=> FLAGS.JIG_Q2_STATUS,
	NEXT_JIG_STATUS:=PMAX_DI.WAGON_WAITING,
	CYLINDER_STOP=> Q2_DO.WAGON_STOP_CYLINDER,
	CYLINDER_LOCK=> Q2_DO.WAGON_LOCK_CYLINDER);

JIG_PMAX(
	CARRIER_PRESENT:=PMAX_DI.WAGON_PRESENT ,
	RELEASE_CARRIER:= FLAGS.PMAX_RELEASE_CARRIER,
	STATUS=> FLAGS.JIG_PMAX_STATUS,
	NEXT_JIG_STATUS:=PRINT_DI.WAGON_WAITING,
	CYLINDER_STOP=> PMAX_DO.WAGON_STOP_CYLINDER,
	CYLINDER_LOCK=> PMAX_DO.WAGON_LOCK_CYLINDER);

JIG_PRINT(
	CARRIER_PRESENT:=PRINT_DI.WAGON_PRESENT ,
	RELEASE_CARRIER:= FLAGS.PRINT_RELEASE_CARRIER,
	STATUS=> FLAGS.JIG_PRINT_STATUS,
	NEXT_JIG_STATUS:=0,
	CYLINDER_STOP=> PRINT_DO.WAGON_STOP_CYLINDER,
	CYLINDER_LOCK=> PRINT_DO.WAGON_LOCK_CYLINDER);

(********************************************
*
* Gestion des posages secondaires
*
********************************************)
JIG_VAC_2nd(
CARRIER_PRESENT:=VAC_DI.WAGON_WAITING ,
CARRIER_PRESENT_MAIN_JIG:=VAC_DI.WAGON_PRESENT,
JIG_STATUS:= FLAGS.JIG_VAC_STATUS,
CYLINDER_WAIT=>VAC_DO.WAGON_WAIT_CYLINDER );

JIG_Q1_2nd(
CARRIER_PRESENT:=Q1_DI.WAGON_WAITING ,
CARRIER_PRESENT_MAIN_JIG:=Q1_DI.WAGON_PRESENT,
JIG_STATUS:= FLAGS.JIG_Q1_STATUS,
CYLINDER_WAIT=>Q1_DO.WAGON_WAIT_CYLINDER );

JIG_Q2_2nd(
CARRIER_PRESENT:=Q2_DI.WAGON_WAITING ,
CARRIER_PRESENT_MAIN_JIG:=Q2_DI.WAGON_PRESENT,
JIG_STATUS:= FLAGS.JIG_Q2_STATUS,
CYLINDER_WAIT=>Q2_DO.WAGON_WAIT_CYLINDER );

JIG_PMAX_2nd(
CARRIER_PRESENT:=PMAX_DI.WAGON_WAITING ,
CARRIER_PRESENT_MAIN_JIG:=PMAX_DI.WAGON_PRESENT,
JIG_STATUS:= FLAGS.JIG_PMAX_STATUS,
CYLINDER_WAIT=>PMAX_DO.WAGON_WAIT_CYLINDER );

JIG_PRINT_2nd(
CARRIER_PRESENT:=PRINT_DI.WAGON_WAITING ,
CARRIER_PRESENT_MAIN_JIG:=PRINT_DI.WAGON_PRESENT,
JIG_STATUS:= FLAGS.JIG_PRINT_STATUS,
CYLINDER_WAIT=>PRINT_DO.WAGON_WAIT_CYLINDER );

(**********************************
*
* FBs
*
********************************************)

END_PROGRAM

// ---- POUs/Carriers/JIG.TcPOU
FUNCTION_BLOCK JIG
VAR
	STEP: INT := 0; (* Internal program step *)
	TIMER_RELEASE: TON;
	START_RELEASE_TIMER:BOOL:=FALSE;
END_VAR

VAR_INPUT
	NEXT_JIG_STATUS:BOOL; (*Status of the next jig*)
	CARRIER_PRESENT:BOOL; (*CARRIER IS PRESENT *)
	RELEASE_CARRIER:BOOL; (*Ask the function to release the carrier *)
END_VAR

VAR_OUTPUT
	STATUS: BOOL := FALSE; (* 0-> JIG FREE   1-> JIB BUSY *)
	CYLINDER_STOP: BOOL :=TRUE; (* STOP the carrier at this position *)
	CYLINDER_LOCK: BOOL:=FALSE; (* LOCK the carrier at this position *)
END_VAR

(************************************************************************************************************************************
*
* Gère le posage principale pour une station (Palette et convoyeur)
*
*
************************************************************************************************************************************)
IF GEMMA.STEP='A6' OR GEMMA.STEP='D1' THEN
	STEP:=0;

END_IF;

CASE STEP OF

0: (*Init*)
	STEP:=STEP+1;
	STATUS:=0;
	START_RELEASE_TIMER:=FALSE;
	CYLINDER_STOP:=TRUE;
	CYLINDER_LOCK:=FALSE;

1: (*Wait for a carrier*)
	IF CARRIER_PRESENT THEN
		CYLINDER_LOCK:=1;
		STATUS:=1;
		STEP:=STEP+1;
	END_IF;

2: (*Release the carrier*)
	IF RELEASE_CARRIER AND NEXT_JIG_STATUS=0 THEN
		CYLINDER_LOCK:=0;
		CYLINDER_STOP:=0;
		START_RELEASE_TIMER:=1;
		STEP:=STEP+1;
	END_IF;

3: (*Delay after release of the carrier*)
	IF TIMER_RELEASE.Q THEN
		CYLINDER_STOP:=1;
		START_RELEASE_TIMER:=0;
		STATUS:=0;
		STEP:=1;
	END_IF;


ELSE
    ;
END_CASE;


(* TIMERS*)
TIMER_RELEASE(IN:=START_RELEASE_TIMER,PT:=CARRIER_RELEASE_DELAY);

END_FUNCTION_BLOCK

// ---- POUs/Carriers/JIG_2ND.TcPOU
FUNCTION_BLOCK JIG_2ND
VAR
	STEP: INT := 0; (* Internal program step *)
	TIMER_STOP: TON;
	R_TRIG1:R_TRIG;
	START_RELEASE_TIMER:BOOL:=FALSE;
	STATUS: BOOL := 0;
END_VAR

VAR_INPUT
	CARRIER_PRESENT:BOOL; (*CARRIER IS PRESENT *)
	CARRIER_PRESENT_MAIN_JIG:BOOL;
	JIG_STATUS:BOOL;
END_VAR

VAR_OUTPUT
	CYLINDER_WAIT: BOOL :=TRUE; (* STOP the carrier at this position *)
END_VAR

(************************************************************************************************************************************
*
* Gère le posage d'attente pour une station (Palette et convoyeur)
*
*
************************************************************************************************************************************)
IF GEMMA.STEP='A6' THEN
	STEP:=0;
END_IF;

CASE STEP OF

0: (*Init*)
	STEP:=STEP+1;
	STATUS:=0;
	START_RELEASE_TIMER:=FALSE;
	CYLINDER_WAIT:=FALSE;

1: (*Wait for a carrier*)
	IF  JIG_STATUS=0 THEN
		CYLINDER_WAIT:=0;
		STEP:=STEP+1;
	END_IF;

2: (*start lock delay*)
	IF  R_TRIG1.Q THEN
		START_RELEASE_TIMER:=1;
		STEP:=STEP+1;
	END_IF;

3: (*Wait the delay before stop the next carrier*)
	IF TIMER_STOP.Q THEN
		CYLINDER_WAIT:=1;
		STEP:=1;
	END_IF;


ELSE 
    ;
END_CASE;

(* TIMERS*)
TIMER_STOP(IN:=START_RELEASE_TIMER,PT:=CARRIER_STOP_DELAY);
R_TRIG1(CLK:= CARRIER_PRESENT_MAIN_JIG);

END_FUNCTION_BLOCK

// ---- POUs/Stations/VAC.TcPOU
PROGRAM VAC
VAR
	STEP: INT := 0;
	R_TRIG1:R_TRIG;
	Suction_Delay: TON;
	FlowStop_Delay: TON;
	Start_FlowStop_Delay: BOOL;
	Pump_Delay: TON;
	Start_Pump_Delay: BOOL;
	Start_Suction_Delay: BOOL;
END_VAR

(*******************************************************
*
* Program fro the PRINT Test station
*
*
*********************************************************)
IF GEMMA.STEP='A6' THEN
	STEP:=0;
END_IF;


CASE STEP OF

0: (*Init*)
	Start_Pump_Delay:=FALSE;
	Start_Suction_Delay:=FALSE;
	Start_FlowStop_Delay:=FALSE;
	FLAGS.VAC_STATUS:=0;
	FLAGS.VAC_RELEASE_CARRIER:=0;
	STEP := STEP+10;

10: (*Wait main JIG Ready*)
	IF R_TRIG1.Q AND GEMMA.STEP='F1'  THEN
		FLAGS.VAC_STATUS:=1;
		STEP := STEP+10;

	END_IF;

20: (*Continue if doors closed**************************************************************************)
	IF FLAGS.DOORS_OPEN=0 THEN
		STEP := STEP+10;
	END_IF;

30: (* Check hydraulique connexion OK*)
	VAC_DO.HYDRO_CYLINDER_BOT:=TRUE;
	VAC_DO.HYDRO_CYLINDER_TOP:=TRUE;

	STEP := STEP+10;

40: (*Continue if doors closed**************************************************************************)
	IF FLAGS.DOORS_OPEN=0 THEN
		STEP := STEP+10;
	END_IF;

50: (* Wait hydraulique connexion OK*)
	IF VAC_DI.CYLINDER_BOT_OUT AND VAC_DI.CYLINDER_TOP_OUT THEN
		STEP := STEP+10;
	END_IF;

60: (*Continue if doors closed**************************************************************************)
	IF FLAGS.DOORS_OPEN=0 THEN
		STEP := STEP+10;
	END_IF;

70: (*Close electrical connexion *)
	VAC_DO.ELECTR_CYLINDER:=TRUE;
	STEP := STEP+10;

80: (*Continue if doors closed**************************************************************************)
	IF FLAGS.DOORS_OPEN=0 THEN
		STEP := STEP+10;
	END_IF;

90:(*Wait electrical connexion closed*)
	IF VAC_DI.POWER_CYLINDER_OUT THEN
		Start_Pump_Delay:=TRUE;
		VAC_DO.PUMP_POWER:=TRUE;
		VAC_DO.FLOW_STOP_VALVE:=TRUE;
		VAC_DO.VACUUM_VALVE:=TRUE;
		STEP := STEP+10;
	END_IF;

100: (*Continue if doors closed**************************************************************************)
	IF FLAGS.DOORS_OPEN=0 THEN
		STEP := STEP+10;
	END_IF;

110: (*Pump until end of delay*)
	IF Pump_Delay.Q THEN
		VAC_DO.VACUUM_VALVE:=FALSE;
		Start_Pump_Delay:=FALSE;
		Start_Suction_Delay:=TRUE;
		STEP := STEP+10;
	END_IF;

120: (*Continue if doors closed**************************************************************************)
	IF FLAGS.DOORS_OPEN=0 THEN
		STEP := STEP+10;
	END_IF;


130: (*Suction until end of delay*)
	IF Suction_Delay.Q THEN
		VAC_DO.HYDRO_CYLINDER_BOT:=FALSE;
		Start_Suction_Delay:=FALSE;
		Start_FlowStop_Delay:=TRUE;
		STEP := STEP+10;
	END_IF;

140: (*Continue if doors closed**************************************************************************)
	IF FLAGS.DOORS_OPEN=0 THEN
		STEP := STEP+10;
	END_IF;

150: (*Delay before FLOWSTOP*)
	IF FlowStop_Delay.Q THEN
		VAC_DO.FLOW_STOP_VALVE:=FALSE;
		VAC_DO.PUMP_POWER:=FALSE;
		Start_FlowStop_Delay:=FALSE;
		STEP := STEP+10;
	END_IF;


160: (*Continue if doors closed**************************************************************************)
	IF FLAGS.DOORS_OPEN=0 THEN
		STEP := STEP+10;
	END_IF;


170: (*Release electrical and hydraulic connexion*)


	VAC_DO.HYDRO_CYLINDER_TOP:=FALSE;
	VAC_DO.ELECTR_CYLINDER:=FALSE;

	STEP := STEP+10;

180: (*Continue if doors closed**************************************************************************)
	IF FLAGS.DOORS_OPEN=0 THEN
		STEP := STEP+10;
	END_IF;

190:(*Wait all cylinders IN*)
	IF VAC_DI.POWER_CYLINDER_IN AND VAC_DI.CYLINDER_BOT_IN AND VAC_DI.CYLINDER_TOP_IN THEN
		STEP := STEP+10;
	END_IF;

200: (*Continue if doors closed**************************************************************************)
	IF FLAGS.DOORS_OPEN=0 THEN
		STEP := STEP+10;
	END_IF;

210: (*Release carrier*)
	FLAGS.VAC_RELEASE_CARRIER:=TRUE;
	STEP:=STEP+10;

220: (*Continue if doors closed**************************************************************************)
	IF FLAGS.DOORS_OPEN=0 THEN
		STEP := STEP+10;
	END_IF;

230: (*Wait carrier away*)
	IF VAC_DI.WAGON_AWAY THEN
		STEP := 0;
	END_IF;



ELSE
    ;
END_CASE;

PROG_STEPS.VAC_STEP:=STEP;

(*FBs*)
Pump_Delay(IN:= Start_Pump_Delay, PT:= PUMP_PARAMS.PMAX_PUMPING_TIME);
Suction_Delay(IN:= Start_Suction_Delay, PT:= PUMP_PARAMS.PMAX_MEASUREMENT_TIME);
FlowStop_Delay(IN:= Start_FlowStop_Delay, PT:= DRY_DELAY);

R_TRIG1(CLK:= CONVEYOR.JIG_VAC.STATUS);

END_PROGRAM

// ---- POUs/Stations/Q1.TcPOU
PROGRAM Q1
VAR
	STEP: INT := 0;
	R_TRIG1:R_TRIG;
	FlowStop_Delay: TON;
	Start_FlowStop_Delay: BOOL;
	Pump_Delay: TON;
	Start_Pump_Delay: BOOL;
	Start_Suction_Delay: BOOL;
	Measurement_Delay: TON;
	Start_Measurement_Delay: BOOL;
	Init_Mass:REAL;

	FB_FormatString1: FB_FormatString;
	sInsertString: STRING;
	bError: BOOL;
	nErrid: DWORD;
	bBusyInsert: BOOL;
	bErrInsert: BOOL;
	nErridInsert: DWORD;
	FB_FormatStringDateTime: FB_FormatString;
	NT_GetTime1: NT_GetTime;
	tTime: TIMESTRUCT;
	bTimestart: BOOL:=0;
	sDateTimeString: T_MaxString;
	bExec_DBRecordInsert1: BOOL;
	P_ERREUR: REAL;
END_VAR

(*******************************************************
*
* Program fro the Q1 Test station
*
*
*********************************************************)
IF GEMMA.STEP='A6' THEN
	STEP:=0;
END_IF;


CASE STEP OF

0: (*Init*)
	Start_Pump_Delay:=FALSE;
	Start_FlowStop_Delay:=FALSE;
	Start_Measurement_Delay:=FALSE;
	Q1_DO.MAX_FLOW_VALVE:=FALSE;
	FLAGS.Q1_STATUS:=0;
	FLAGS.Q1_RELEASE_CARRIER:=0;
	Q1_FLOWMETER_CONTROL.SET_TOT:=1; (*Reset mass flow counter*)
	STEP := STEP+10;

10: (*Wait main JIG Ready*)
	IF R_TRIG1.Q AND GEMMA.STEP='F1'  THEN
		FLAGS.Q1_STATUS:=1;
		Q1_FLOWMETER_CONTROL.SET_TOT:=0; (*Reset mass flow counter*)
		Q1_CALCULETED_FLOW:=0;
		STEP := STEP+10;
	END_IF;

20: (*Continue if doors closed**************************************************************************)
	IF FLAGS.DOORS_OPEN=0 THEN
		STEP := STEP+10;
	END_IF;

30: (* Check hydraulique connexion OK*)
	Q1_DO.HYDRO_CYLINDER_BOT:=TRUE;
	Q1_DO.HYDRO_CYLINDER_TOP:=TRUE;


	STEP := STEP+10;

40: (*Continue if doors closed**************************************************************************)
	IF FLAGS.DOORS_OPEN=0 THEN
		STEP := STEP+10;
	END_IF;

50: (* Wait hydraulique connexion OK*)
	IF Q1_DI.CYLINDER_BOT_OUT AND Q1_DI.CYLINDER_TOP_OUT THEN
		STEP := STEP+10;
	END_IF;

60: (*Continue if doors closed**************************************************************************)
	IF FLAGS.DOORS_OPEN=0 THEN
		STEP := STEP+10;
	END_IF;

70: (*Close electrical connexion *)
	Q1_DO.ELECTR_CYLINDER:=TRUE;
	Q1_DO.MAX_FLOW_VALVE:=TRUE;
	STEP := STEP+10;

80: (*Continue if doors closed**************************************************************************)
	IF FLAGS.DOORS_OPEN=0 THEN
		STEP := STEP+10;
	END_IF;

90:(*Wait electrical connexion closed*)
	IF Q1_DI.POWER_CYLINDER_OUT THEN
		Start_Pump_Delay:=TRUE;
		(*Q1_DO.MAX_FLOW_VALVE:=PUMP_PARAMS.Q1_MAX_FLOW;*)
		Q1_DO.MAX_FLOW_VALVE:=TRUE;
		Q1_DO.PUMP_POWER:=TRUE;
		Q1_DO.FLOW_STOP_VALVE:=TRUE;
		Q1_DO.FLOW_STOP_BOTT:=TRUE;
		STEP := STEP+10;
	END_IF;

100: (*Continue if doors closed**************************************************************************)
	IF FLAGS.DOORS_OPEN=0 THEN
		STEP := STEP+10;
	END_IF;

110: (*Pump until end of delay*)

	(*Regulation de la pression pendant le temps d'amorcage et ne bouge plus pendant le temps de mesure*)
	(* Regulation seulement à +- 20% de la consigne et seulement après X secondes*)
	IF  Pump_Delay.ET>T#15s AND Q1_FLOWMETER_VALUES.VolumeFlow>50 THEN
				Q1_DO.MAX_FLOW_VALVE:=FALSE;
				P_ERREUR:=PUMP_PARAMS.Q1_PRESSURE_TARGET - Q1_PRESSURE_SENSOR_VALUE;
				FLAGS.MOTOR_Q1_POSITION := FLAGS.MOTOR_Q1_POSITION + REAL_TO_INT(P_ERREUR*7);(* P_ERREUR*GAIN *)
	END_IF


	IF Pump_Delay.Q THEN
		Start_Pump_Delay:=FALSE;
		Start_Measurement_Delay:=TRUE;
		Init_Mass:=Q1_FLOWMETER_VALUES.TotalMass; (*Store the mass at the beginning of the measurement*)
		STEP := STEP+10;
	END_IF;

120: (*Continue if doors closed**************************************************************************)
	IF FLAGS.DOORS_OPEN=0 THEN
		STEP := STEP+10;
	END_IF;


130: (*Measurement delay*)

	(*test*)
	IF 		(Q1_PRESSURE_SENSOR_VALUE<PUMP_PARAMS.Q1_PRESSURE_TARGET+10)
			AND (Q1_PRESSURE_SENSOR_VALUE>PUMP_PARAMS.Q1_PRESSURE_TARGET-10)
			AND Q1_FLOWMETER_VALUES.VolumeFlow>50 THEN

				P_ERREUR:=PUMP_PARAMS.Q1_PRESSURE_TARGET - Q1_PRESSURE_SENSOR_VALUE;
				FLAGS.MOTOR_Q1_POSITION := FLAGS.MOTOR_Q1_POSITION + REAL_TO_INT(P_ERREUR*7);(* P_ERREUR*GAIN *)
	END_IF
	(*end test*)

	IF Measurement_Delay.Q THEN
		Q1_CALCULETED_FLOW:=CONVERT_MASS_TO_FLOW(Q1_FLOWMETER_VALUES.TotalMass-Init_Mass, PUMP_PARAMS.Q1_MEASUREMENT_TIME); (*Convert mass to massflow*)
		Q1_DO.HYDRO_CYLINDER_BOT:=FALSE;
		Q1_DO.MAX_FLOW_VALVE:=TRUE;
		Start_Measurement_Delay:=FALSE;
		Start_FlowStop_Delay:=TRUE;
		STEP := STEP+10;
	END_IF;


140: (*Continue if doors closed**************************************************************************)
	IF FLAGS.DOORS_OPEN=0 THEN
		STEP := STEP+10;
	END_IF;


150: (*Delay before FLOWSTOP*)
	IF FlowStop_Delay.Q THEN
		Q1_DO.FLOW_STOP_VALVE:=FALSE;
		Q1_DO.MAX_FLOW_VALVE:=FALSE;
		Q1_DO.FLOW_STOP_BOTT:=FALSE;
		Q1_DO.PUMP_POWER:=FALSE;
		Start_FlowStop_Delay:=FALSE;
		bExec_DBRecordInsert1:=FALSE; (*Deactivate DB Record*)
		STEP := STEP+10;
	END_IF;


160: (*Continue if doors closed**************************************************************************)
	IF FLAGS.DOORS_OPEN=0 THEN
		STEP := STEP+10;
	END_IF;


170: (*Release electrical and hydraulic connexion*)

	Q1_DO.ELECTR_CYLINDER:=FALSE;
	Q1_DO.HYDRO_CYLINDER_TOP:=FALSE;

	STEP := STEP+10;

180: (*Continue if doors closed**************************************************************************)
	IF FLAGS.DOORS_OPEN=0 THEN
		STEP := STEP+10;
	END_IF;

190:(*Wait all cylinders IN*)
	IF Q1_DI.POWER_CYLINDER_IN AND Q1_DI.CYLINDER_TOP_IN AND Q1_DI.CYLINDER_BOT_IN THEN
		STEP := STEP+10;
	END_IF;

200: (*Continue if doors closed**************************************************************************)
	IF FLAGS.DOORS_OPEN=0 THEN
		STEP := STEP+10;
	END_IF;

210: (*Release carrier*)
	FLAGS.Q1_RELEASE_CARRIER:=TRUE;
	STEP:=STEP+10;

220: (*Continue if doors closed**************************************************************************)
	IF FLAGS.DOORS_OPEN=0 THEN
		STEP := STEP+10;
	END_IF;

230: (*Wait carrier away*)
	IF Q1_DI.WAGON_AWAY THEN
		STEP := 0;
	END_IF;



ELSE
    ;
END_CASE;

(*FBs*)
Pump_Delay(IN:= Start_Pump_Delay, PT:= PUMP_PARAMS.Q1_PUMPING_TIME);

Measurement_Delay(IN:= Start_Measurement_Delay, PT:= PUMP_PARAMS.Q1_MEASUREMENT_TIME);

FlowStop_Delay(IN:= Start_FlowStop_Delay, PT:=DRY_DELAY);

R_TRIG1(CLK:= CONVEYOR.JIG_Q1.STATUS);

PROG_STEPS.Q1_STEP:=STEP;

END_PROGRAM

// ---- POUs/Functions/CONVERT_MASS_TO_FLOW.TcPOU
FUNCTION CONVERT_MASS_TO_FLOW : REAL
VAR_INPUT
	Mass:REAL; (*in gramme*)
	Delay:TIME; (*in ms*)
END_VAR
VAR
END_VAR

CONVERT_MASS_TO_FLOW:=Mass/TIME_TO_DWORD(Delay)*60000;

END_FUNCTION

// ---- POUs/Stations/Q2.TcPOU
PROGRAM Q2
VAR
	STEP: INT := 0;
	R_TRIG1:R_TRIG;
	FlowStop_Delay: TON;
	Start_FlowStop_Delay: BOOL;
	Pump_Delay: TON;
	Start_Pump_Delay: BOOL;
	Start_Suction_Delay: BOOL;
	Measurement_Delay: TON;
	Start_Measurement_Delay: BOOL;
	Init_Mass:REAL;

	FB_FormatString1: FB_FormatString;
	sInsertString: STRING;
	bError: BOOL;
	nErrid: DWORD;
	bBusyInsert: BOOL;
	bErrInsert: BOOL;
	nErridInsert: DWORD;
	FB_FormatStringDateTime: FB_FormatString;
	NT_GetTime1: NT_GetTime;
	tTime: TIMESTRUCT;
	bTimestart: BOOL:=0;
	sDateTimeString: T_MaxString;
	bExec_DBRecordInsert1: BOOL;
	P_ERREUR: REAL;
END_VAR

(*******************************************************
*
* Program fro the Q2 Test station
*
*
*********************************************************)
IF GEMMA.STEP='A6' THEN
	STEP:=0;
END_IF;


CASE STEP OF

0: (*Init*)
	Start_Pump_Delay:=FALSE;
	Start_FlowStop_Delay:=FALSE;
	Start_Measurement_Delay:=FALSE;
	Q2_DO.MAX_FLOW_VALVE:=FALSE;
	FLAGS.Q2_STATUS:=0;
	FLAGS.Q2_RELEASE_CARRIER:=0;
	Q2_FLOWMETER_CONTROL.SET_TOT:=1; (*Reset mass flow counter*)
	STEP := STEP+10;

10: (*Wait main JIG Ready*)
	IF R_TRIG1.Q AND GEMMA.STEP='F1'  THEN
		FLAGS.Q2_STATUS:=1;
		Q2_FLOWMETER_CONTROL.SET_TOT:=0; (*Reset mass flow counter*)
		Q2_CALCULETED_FLOW:=0;
		STEP := STEP+10;
	END_IF;

20: (*Continue if doors closed**************************************************************************)
	IF FLAGS.DOORS_OPEN=0 THEN
		STEP := STEP+10;
	END_IF;

30: (* Check hydraulique connexion OK*)
	Q2_DO.HYDRO_CYLINDER_BOT:=TRUE;
	Q2_DO.HYDRO_CYLINDER_TOP:=TRUE;


	STEP := STEP+10;

40: (*Continue if doors closed**************************************************************************)
	IF FLAGS.DOORS_OPEN=0 THEN
		STEP := STEP+10;
	END_IF;

50: (* Wait hydraulique connexion OK*)
	IF Q2_DI.CYLINDER_BOT_OUT AND Q2_DI.CYLINDER_TOP_OUT THEN
		STEP := STEP+10;
	END_IF;

60: (*Continue if doors closed**************************************************************************)
	IF FLAGS.DOORS_OPEN=0 THEN
		STEP := STEP+10;
	END_IF;

70: (*Close electrical connexion *)
	Q2_DO.ELECTR_CYLINDER:=TRUE;
	Q2_DO.MAX_FLOW_VALVE:=TRUE;
	STEP := STEP+10;

80: (*Continue if doors closed**************************************************************************)
	IF FLAGS.DOORS_OPEN=0 THEN
		STEP := STEP+10;
	END_IF;

90:(*Wait electrical connexion closed*)
	IF Q2_DI.POWER_CYLINDER_OUT THEN
		Start_Pump_Delay:=TRUE;
		(*Q2_DO.MAX_FLOW_VALVE:=PUMP_PARAMS.Q2_MAX_FLOW;*)
		Q2_DO.MAX_FLOW_VALVE:=TRUE;
		Q2_DO.PUMP_POWER:=TRUE;
		Q2_DO.FLOW_STOP_VALVE:=TRUE;
		Q2_DO.FLOW_STOP_BOTT:=TRUE;
		STEP := STEP+10;
	END_IF;

100: (*Continue if doors closed**************************************************************************)
	IF FLAGS.DOORS_OPEN=0 THEN
		STEP := STEP+10;
	END_IF;

110: (*Pump until end of delay*)



	(*Regulation de la pression pendant le temps d'amorcage et ne bouge plus pendant le temps de mesure*)
	(* Regulation seulement à +- 20% de la consigne et seulement après X secondes*)
	(*IF 		(Q2_PRESSURE_SENSOR_VALUE<PUMP_PARAMS.Q2_PRESSURE_TARGET+10)
			AND (Q2_PRESSURE_SENSOR_VALUE>PUMP_PARAMS.Q2_PRESSURE_TARGET-10)
			AND Pump_Delay.ET>T#10s THEN

				P_ERREUR:=PUMP_PARAMS.Q2_PRESSURE_TARGET - Q2_PRESSURE_SENSOR_VALUE;
				FLAGS.MOTOR_Q2_POSITION := FLAGS.MOTOR_Q2_POSITION + REAL_TO_INT(P_ERREUR*10);(* P_ERREUR*GAIN *)
	END_IF*)

	IF 		Pump_Delay.ET>T#15s AND Q2_FLOWMETER_VALUES.VolumeFlow>50 THEN
				Q2_DO.MAX_FLOW_VALVE:=FALSE;
				P_ERREUR:=PUMP_PARAMS.Q2_PRESSURE_TARGET - Q2_PRESSURE_SENSOR_VALUE;
				FLAGS.MOTOR_Q2_POSITION := FLAGS.MOTOR_Q2_POSITION + REAL_TO_INT(P_ERREUR*7);(* P_ERREUR*GAIN *)
	END_IF


	IF Pump_Delay.Q THEN
		Start_Pump_Delay:=FALSE;
		Start_Measurement_Delay:=TRUE;
		Init_Mass:=Q2_FLOWMETER_VALUES.TotalMass; (*Store the mass at the beginning of the measurement*)
		STEP := STEP+10;
	END_IF;

120: (*Continue if doors closed**************************************************************************)
	IF FLAGS.DOORS_OPEN=0 THEN
		STEP := STEP+10;
	END_IF;


130: (*Measurement delay*)




	IF 		(Q2_PRESSURE_SENSOR_VALUE<PUMP_PARAMS.Q2_PRESSURE_TARGET+10)
			AND (Q2_PRESSURE_SENSOR_VALUE>PUMP_PARAMS.Q2_PRESSURE_TARGET-10)
			AND Q2_FLOWMETER_VALUES.VolumeFlow>50 THEN

				P_ERREUR:=PUMP_PARAMS.Q2_PRESSURE_TARGET - Q2_PRESSURE_SENSOR_VALUE;
				FLAGS.MOTOR_Q2_POSITION := FLAGS.MOTOR_Q2_POSITION + REAL_TO_INT(P_ERREUR*7);(* P_ERREUR*GAIN *)
	END_IF

	IF Measurement_Delay.Q THEN
		Q2_CALCULETED_FLOW:=CONVERT_MASS_TO_FLOW(Q2_FLOWMETER_VALUES.TotalMass-Init_Mass, PUMP_PARAMS.Q2_MEASUREMENT_TIME); (*Convert mass to massflow*)
		Q2_DO.HYDRO_CYLINDER_BOT:=FALSE;
		Q2_DO.MAX_FLOW_VALVE:=TRUE;
		Start_Measurement_Delay:=FALSE;
		Start_FlowStop_Delay:=TRUE;
		STEP := STEP+10;
	END_IF;


140: (*Continue if doors closed**************************************************************************)
	IF FLAGS.DOORS_OPEN=0 THEN
		STEP := STEP+10;
	END_IF;


150: (*Delay before FLOWSTOP*)
	IF FlowStop_Delay.Q THEN
		Q2_DO.FLOW_STOP_VALVE:=FALSE;
		Q2_DO.MAX_FLOW_VALVE:=FALSE;
		Q2_DO.FLOW_STOP_BOTT:=FALSE;
		Q2_DO.PUMP_POWER:=FALSE;
		Start_FlowStop_Delay:=FALSE;
		bExec_DBRecordInsert1:=FALSE; (*Deactivate DB Record*)
		STEP := STEP+10;
	END_IF;


160: (*Continue if doors closed**************************************************************************)
	IF FLAGS.DOORS_OPEN=0 THEN
		STEP := STEP+10;
	END_IF;


170: (*Release electrical and hydraulic connexion*)

	Q2_DO.ELECTR_CYLINDER:=FALSE;
	Q2_DO.HYDRO_CYLINDER_TOP:=FALSE;

	STEP := STEP+10;

180: (*Continue if doors closed**************************************************************************)
	IF FLAGS.DOORS_OPEN=0 THEN
		STEP := STEP+10;
	END_IF;

190:(*Wait all cylinders IN*)
	IF Q2_DI.POWER_CYLINDER_IN AND Q2_DI.CYLINDER_TOP_IN AND Q2_DI.CYLINDER_BOT_IN THEN
		STEP := STEP+10;
	END_IF;

200: (*Continue if doors closed**************************************************************************)
	IF FLAGS.DOORS_OPEN=0 THEN
		STEP := STEP+10;
	END_IF;

210: (*Release carrier*)
	FLAGS.Q2_RELEASE_CARRIER:=TRUE;
	STEP:=STEP+10;

220: (*Continue if doors closed**************************************************************************)
	IF FLAGS.DOORS_OPEN=0 THEN
		STEP := STEP+10;
	END_IF;

230: (*Wait carrier away*)
	IF Q2_DI.WAGON_AWAY THEN
		STEP := 0;
	END_IF;



ELSE
    ;
END_CASE;

(*FBs*)
Pump_Delay(IN:= Start_Pump_Delay, PT:= PUMP_PARAMS.Q2_PUMPING_TIME);

Measurement_Delay(IN:= Start_Measurement_Delay, PT:= PUMP_PARAMS.Q2_MEASUREMENT_TIME);

FlowStop_Delay(IN:= Start_FlowStop_Delay, PT:=DRY_DELAY);

R_TRIG1(CLK:= CONVEYOR.JIG_Q2.STATUS);

PROG_STEPS.Q2_STEP:=STEP;

END_PROGRAM

// ---- POUs/Stations/PRINT.TcPOU
PROGRAM PRINT
VAR
	STEP: INT := 0;
	R_TRIG1:R_TRIG;
	Suction_Delay: TON;
	FlowStop_Delay: TON;
	Start_FlowStop_Delay: BOOL;
	Pump_Delay: TON;
	Start_Pump_Delay: BOOL;
	Start_Suction_Delay: BOOL;
	Start_Step20_Delay: BOOL;
	TON_Step20: TON;
END_VAR

(*******************************************************
*
* Program fro the VACUUM Test station
*
*
*********************************************************)
IF GEMMA.STEP='A6' THEN
	STEP:=0;
END_IF;


CASE STEP OF

0: (*Init*)
	Start_Pump_Delay:=FALSE;
	Start_Suction_Delay:=FALSE;
	Start_FlowStop_Delay:=FALSE;
	Start_Step20_Delay:=FALSE;
	FLAGS.PRINT_STATUS:=0;
	FLAGS.PRINT_RELEASE_CARRIER:=0;
	STEP := STEP+10;

10: (*Wait main JIG Ready*)
	IF R_TRIG1.Q AND GEMMA.STEP='F1'  THEN
		FLAGS.PRINT_STATUS:=1;
		Start_Step20_Delay:=TRUE;
		STEP := STEP+10;

	END_IF;

20: (*Continue if doors closed**************************************************************************)
	IF FLAGS.DOORS_OPEN=0 AND TON_Step20.Q THEN
		STEP := STEP+10;
	END_IF;

	(*Ajouter un délai de 1 secondes*******************************************************************3*)

30: (* Check hydraulique connexion OK*)
	IF PRINT_PUMP_STATUS=FALSE AND NOT(RUN_CG) THEN
		STEP := STEP+10;
	ELSE
		STEP:= 210;
	END_IF

(*************)
40: (* Open Gripper and go down to pick the part*)
	PRINT_DO.EJECTION_GRIPPER:=TRUE;
	PRINT_DO.EJECTION_CYLINDER_Z:=TRUE;
	STEP := STEP+10;

50: (* Wait movement*)
	IF PRINT_DI.GRIPPER_OPEN AND PRINT_DI.Z_DOWN THEN
		PRINT_DO.EJECTION_GRIPPER:=FALSE;
		STEP := STEP+10;
	END_IF

60: (* Wait gripper CLOSED and move UP*)
	IF NOT(PRINT_DI.GRIPPER_OPEN) THEN
		PRINT_DO.EJECTION_CYLINDER_Z:=FALSE;
		STEP := STEP+10;
	END_IF

70: (* Wait movement and move X out*)
	IF PRINT_DI.Z_UP THEN
		PRINT_DO.EJECTION_CYLINDER_X:=TRUE;
		STEP := STEP+10;
	END_IF

80: (* Wait movement and move Z down*)
	IF PRINT_DI.X_OUT THEN
		PRINT_DO.EJECTION_CYLINDER_Z:=TRUE;
		STEP := STEP+10;
	END_IF

90: (* Wait movement and release gripper*)
	IF PRINT_DI.Z_DOWN THEN
		PRINT_DO.EJECTION_GRIPPER:=TRUE;
		STEP := STEP+10;
	END_IF

100: (* Wait gripper open*)
	IF PRINT_DI.GRIPPER_OPEN THEN
		PRINT_DO.EJECTION_CYLINDER_Z:=FALSE;
		STEP := STEP+10;
	END_IF

110: (* Wait movement and go X IN*)
	IF PRINT_DI.Z_UP THEN
		PRINT_DO.EJECTION_CYLINDER_X:=FALSE;
		STEP := STEP + 10;
	END_IF

120: (* Wait movement and go X IN*)
	IF PRINT_DI.X_IN THEN
		STEP := 210;
	END_IF


(**************)

210: (*Release carrier*)
	FLAGS.PRINT_RELEASE_CARRIER:=TRUE;
	STEP:=STEP+10;

220: (*Continue if doors closed**************************************************************************)
	IF FLAGS.DOORS_OPEN=0 THEN
		STEP := STEP+10;
	END_IF;

230: (*Wait carrier away*)
		STEP := 0;




ELSE
    ;
END_CASE;

PROG_STEPS.PRINT_STEP:=STEP;

(*FBs*)

R_TRIG1(CLK:= CONVEYOR.JIG_PRINT.STATUS);
TON_Step20(IN:= Start_Step20_Delay, PT:=T#2s);

END_PROGRAM

// ---- POUs/USB.TcPOU
PROGRAM USB
VAR
END_VAR

;

END_PROGRAM

// ---- POUs/MAIN.TcPOU
PROGRAM MAIN

VAR

END_VAR

GEMMA();
WATER_TANKS();
AIS();
SAFETY();
Q1_MOTOR();
Q2_MOTOR();

END_PROGRAM

// ---- POUs/Water/WATER_TANKS.TcPOU
PROGRAM WATER_TANKS
VAR

	TANK_VAC:WATER_TANK;
	TANK_Q1:WATER_TANK;
	TANK_Q2:WATER_TANK;
	TANK_PMAX:WATER_TANK;



END_VAR
VAR_OUTPUT
	TIMOUT_TANK_VAC: BOOL;
	TIMOUT_TANK_Q1: BOOL;
	TIMOUT_TANK_Q2: BOOL;
	TIMOUT_TANK_PMAX: BOOL;
END_VAR

TANK_VAC(
WATER_TANK_HIGH:= VAC_DI.WATER_TANK_HIGH,
WATER_TANK_LOW:=  VAC_DI.WATER_TANK_LOW,
WATER_TANK_VALVE=> VAC_DO.WATER_TANK_VALVE,
TIMEOUT=> TIMOUT_TANK_VAC
);

TANK_Q1(
WATER_TANK_HIGH:= Q1_DI.WATER_TANK_HIGH,
WATER_TANK_LOW:=  Q1_DI.WATER_TANK_LOW,
WATER_TANK_VALVE=> Q1_DO.WATER_TANK_VALVE,
TIMEOUT=> TIMOUT_TANK_Q1
);


TANK_Q2(
WATER_TANK_HIGH:= Q2_DI.WATER_TANK_HIGH,
WATER_TANK_LOW:=  Q2_DI.WATER_TANK_LOW,
WATER_TANK_VALVE=> Q2_DO.WATER_TANK_VALVE,
TIMEOUT=> TIMOUT_TANK_Q2
);

TANK_PMAX(
WATER_TANK_HIGH:= PMAX_DI.WATER_TANK_HIGH,
WATER_TANK_LOW:=  PMAX_DI.WATER_TANK_LOW,
WATER_TANK_VALVE=> PMAX_DO.WATER_TANK_VALVE,
TIMEOUT=> TIMOUT_TANK_PMAX
);

END_PROGRAM

// ---- POUs/Water/WATER_TANK.TcPOU
FUNCTION_BLOCK WATER_TANK

VAR_INPUT
	WATER_TANK_HIGH: BOOL;
	WATER_TANK_LOW: BOOL;
END_VAR

VAR_OUTPUT
	WATER_TANK_VALVE:BOOL;
	TIMEOUT:BOOL;
END_VAR

VAR
	SR1:SR;
	TON1:TON;
END_VAR

(********************************************************
*
* Water Tank
*
***********************************************************)

SR1(SET1:= NOT WATER_TANK_LOW , RESET:= WATER_TANK_HIGH );

TON1(IN:= SR1.Q1, PT:= TIMEOUT_WATER_TANK);

TIMEOUT:= TON1.Q;

IF SR1.Q1 AND NOT TIMEOUT THEN
	WATER_TANK_VALVE:=TRUE;
ELSE
	WATER_TANK_VALVE:=FALSE;
END_IF;

END_FUNCTION_BLOCK

// ---- POUs/AIS.TcPOU
PROGRAM AIS
VAR
	VAC_SENSOR_VAC_CONVERT: WIKA_GET_VALUES;
	P_SENSOR_Q1_CONVERT: WIKA_GET_VALUES;
	FLOW_SENSOR_Q1_CONVERT: EH_FLOMETER;
	P_SENSOR_Q2_CONVERT: WIKA_GET_VALUES;
	P_SENSOR_PMAX_CONVERT: WIKA_GET_VALUES;
	FLOW_SENSOR_Q2_CONVERT: EH_FLOMETER;
END_VAR

(**********************************************************************
*
*Conversion des entrées analogiques
*
*
*************************************************************************)

(*VAC***************************************************************************)
VAC_SENSOR_VAC_CONVERT(
INPUTS:= VAC_VACUUM_SENSOR.VALUE,
Pressure=> VAC_VACUMM_SENSOR_VALUE);


(*Q1***************************************************************************)
FLOW_SENSOR_Q1_CONVERT(
	AI1:= Q1_FLOWMETER.A1,
	AI2:= Q1_FLOWMETER.A2,
	AI3:= Q1_FLOWMETER.A3,
	AI4:= Q1_FLOWMETER.A4,
	AI5:= Q1_FLOWMETER.A5,
	AI6:= Q1_FLOWMETER.A6,
	TOT:= Q1_FLOWMETER.TOT,
	MassFlow=> Q1_FLOWMETER_VALUES.MassFlow,
	VolumeFlow=> Q1_FLOWMETER_VALUES.VolumeFlow,
	CorrectedVolueFLow=> Q1_FLOWMETER_VALUES.CorrectedVolueFLow,
	Density=> Q1_FLOWMETER_VALUES.Density,
	ReferenceDensity=> Q1_FLOWMETER_VALUES.ReferenceDensity,
	Temperature=> Q1_FLOWMETER_VALUES.Temperature,
	TotalMass=>Q1_FLOWMETER_VALUES.TotalMass);

P_SENSOR_Q1_CONVERT(
INPUTS:= Q1_PRESSURE_SENSOR.VALUE,
Pressure=> Q1_PRESSURE_SENSOR_VALUE);

Q1_CURRENT:=Q1_Multimeter_value/1000.0;

(*Q2***************************************************************************)
FLOW_SENSOR_Q2_CONVERT(
	AI1:= Q2_FLOWMETER.A1,
	AI2:= Q2_FLOWMETER.A2,
	AI3:= Q2_FLOWMETER.A3,
	AI4:= Q2_FLOWMETER.A4,
	AI5:= Q2_FLOWMETER.A5,
	AI6:= Q2_FLOWMETER.A6,
	TOT:= Q2_FLOWMETER.TOT,
	MassFlow=> Q2_FLOWMETER_VALUES.MassFlow,
	VolumeFlow=> Q2_FLOWMETER_VALUES.VolumeFlow,
	CorrectedVolueFLow=> Q2_FLOWMETER_VALUES.CorrectedVolueFLow,
	Density=> Q2_FLOWMETER_VALUES.Density,
	ReferenceDensity=> Q2_FLOWMETER_VALUES.ReferenceDensity,
	Temperature=> Q2_FLOWMETER_VALUES.Temperature,
	TotalMass=>Q2_FLOWMETER_VALUES.TotalMass);

P_SENSOR_Q2_CONVERT(
INPUTS:= Q2_PRESSURE_SENSOR.VALUE,
Pressure=> Q2_PRESSURE_SENSOR_VALUE);

Q2_CURRENT:=Q2_Multimeter_value/1000.0;

(*PMAX***************************************************************************)

P_SENSOR_PMAX_CONVERT(
INPUTS:= PMAX_PRESSURE_SENSOR.VALUE,
Pressure=> PMAX_PRESSURE_SENSOR_VALUE);

END_PROGRAM

// ---- POUs/WIKA/WIKA_GET_VALUES.TcPOU
FUNCTION_BLOCK WIKA_GET_VALUES

VAR_INPUT
	INPUTS: ARRAY [0..7] OF USINT;
END_VAR

VAR_OUTPUT
	Pressure: REAL;
	Measuring_Type:BOOL; (*0->Relativ 1->Absolute*)
END_VAR

VAR
	Pressure_Value:REAL;
	Sign:SINT;
	Sign_Exponent:INT;
	Exponent:REAL;
END_VAR

Pressure_Value:= 	BOOL_TO_INT(INPUTS[1].0)*1 +
			BOOL_TO_INT(INPUTS[1].1)*2 +
			BOOL_TO_INT(INPUTS[1].2)*4 +
			BOOL_TO_INT(INPUTS[1].3)*8 +
			BOOL_TO_INT(INPUTS[1].4)*16 +
			BOOL_TO_INT(INPUTS[1].5)*32 +
			BOOL_TO_INT(INPUTS[1].6)*64 +
			BOOL_TO_INT(INPUTS[1].7)*128+
			BOOL_TO_INT(INPUTS[0].0)*256 +
			BOOL_TO_INT(INPUTS[0].1)*512 +
			BOOL_TO_INT(INPUTS[0].2)*1024 +
			BOOL_TO_INT(INPUTS[0].3)*2048 +
			BOOL_TO_INT(INPUTS[0].4)*4096 +
			BOOL_TO_INT(INPUTS[0].5)*8192 +
			BOOL_TO_INT(INPUTS[0].6)*16384;

IF INPUTS[0].7=0 THEN
Sign:=1;
ELSE
Sign:=-1;
END_IF

Measuring_Type:=INPUTS[2].7;

Sign_Exponent:=BOOL_TO_SINT(INPUTS[2].6)*-1;

Exponent:=	EXPT(10,(BOOL_TO_INT(INPUTS[2].3)*1 + BOOL_TO_INT(INPUTS[2].4)*2 + BOOL_TO_INT(INPUTS[2].5)*4)*Sign_Exponent);

Pressure:=Exponent*Pressure_Value*Sign;

END_FUNCTION_BLOCK

// ---- POUs/EH/EH_FLOMETER.TcPOU
FUNCTION_BLOCK EH_FLOMETER

VAR_INPUT
	AI1: ARRAY [0..4] OF USINT;
	AI2: ARRAY [0..4] OF USINT;
	AI3: ARRAY [0..4] OF USINT;
	AI4: ARRAY [0..4] OF USINT;
	AI5: ARRAY [0..4] OF USINT;
	AI6: ARRAY [0..4] OF USINT;
	TOT: ARRAY [0..4] OF USINT;
END_VAR

VAR_OUTPUT
	MassFlow: REAL;
	VolumeFlow: REAL;
	CorrectedVolueFLow: REAL;
	Density: REAL;
	ReferenceDensity:REAL;
	Temperature:REAL;
	TotalMass: REAL;
END_VAR

VAR

END_VAR

MassFlow:=EH_IEEE754_TO_REAL(AI1);
VolumeFlow:=EH_IEEE754_TO_REAL(AI2);
CorrectedVolueFLow:=EH_IEEE754_TO_REAL(AI3);
Density:=EH_IEEE754_TO_REAL(AI4);
ReferenceDensity:=EH_IEEE754_TO_REAL(AI5);
Temperature:=EH_IEEE754_TO_REAL(AI6);
TotalMass:=EH_IEEE754_TO_REAL(TOT);

END_FUNCTION_BLOCK

// ---- POUs/EH/EH_IEEE754_TO_REAL.TcPOU
FUNCTION EH_IEEE754_TO_REAL : REAL
VAR_INPUT
	AI: ARRAY [0..4] OF USINT;
END_VAR

VAR
	Sign: SINT;
	Exponent:INT;
	Mantisse: REAL;
END_VAR

Sign:=		BOOL_TO_SINT(AI[0].7)*-1;

Exponent:= 	BOOL_TO_SINT(AI[1].7)*1 +
			BOOL_TO_SINT(AI[0].0)*2 +
			BOOL_TO_SINT(AI[0].1)*4 +
			BOOL_TO_SINT(AI[0].2)*8 +
			BOOL_TO_SINT(AI[0].3)*16 +
			BOOL_TO_SINT(AI[0].4)*32 +
			BOOL_TO_SINT(AI[0].5)*64 +
			BOOL_TO_SINT(AI[0].6)*128;

(*met à zéro le bit 7 du byte 1 qui n'est pas dans le mantisse*)
AI[1].7:=0;

Mantisse:=	BOOL_TO_SINT(AI[1].0)*EXPT(2,-7) +
			BOOL_TO_SINT(AI[1].1)*EXPT(2,-6) +
			BOOL_TO_SINT(AI[1].2)*EXPT(2,-5) +
			BOOL_TO_SINT(AI[1].3)*EXPT(2,-4) +
			BOOL_TO_SINT(AI[1].4)*EXPT(2,-3) +
			BOOL_TO_SINT(AI[1].5)*EXPT(2,-2) +
			BOOL_TO_SINT(AI[1].6)*EXPT(2,-1) +
			BOOL_TO_SINT(AI[2].0)*EXPT(2,-15) +
			BOOL_TO_SINT(AI[2].1)*EXPT(2,-14) +
			BOOL_TO_SINT(AI[2].2)*EXPT(2,-13) +
			BOOL_TO_SINT(AI[2].3)*EXPT(2,-12) +
			BOOL_TO_SINT(AI[2].4)*EXPT(2,-11) +
			BOOL_TO_SINT(AI[2].5)*EXPT(2,-10) +
			BOOL_TO_SINT(AI[2].6)*EXPT(2,-9) +
			BOOL_TO_SINT(AI[2].7)*EXPT(2,-8) +
			BOOL_TO_SINT(AI[3].0)*EXPT(2,-23) +
			BOOL_TO_SINT(AI[3].1)*EXPT(2,-22) +
			BOOL_TO_SINT(AI[3].2)*EXPT(2,-21) +
			BOOL_TO_SINT(AI[3].3)*EXPT(2,-20) +
			BOOL_TO_SINT(AI[3].4)*EXPT(2,-19) +
			BOOL_TO_SINT(AI[3].5)*EXPT(2,-18) +
			BOOL_TO_SINT(AI[3].6)*EXPT(2,-17) +
			BOOL_TO_SINT(AI[3].7)*EXPT(2,-16);

EH_IEEE754_TO_REAL:=EXPT(-1,Sign)*EXPT(2,Exponent-127)*(1+Mantisse);

IF EH_IEEE754_TO_REAL<0.000001 THEN
EH_IEEE754_TO_REAL:=0;
END_IF;

END_FUNCTION

// ---- POUs/SAFETY.TcPOU
PROGRAM SAFETY
VAR
END_VAR

SAFETY_OUT.DOORS_RUN:=TRUE;

SAFETY_OUT.DOORS_ErrAck:=SAFETY_OUT.NOT_AUS_RESET;


IF SAFETY_IN.NOT_AUS_State=1 THEN

	FLAGS.SAFETY_OK:=TRUE;

ELSE

	FLAGS.SAFETY_OK:=FALSE;
END_IF;

END_PROGRAM

// ---- POUs/Q1_MOTOR.TcPOU
PROGRAM Q1_MOTOR
VAR
	ClearFault: FB_ClearFault;
	SetEnableState: FB_SetEnableState;
	SetHomingParameter: FB_SetHomingParameter;
	FindHome: FB_FindHome;
	SetMotorParameter: FB_SetMotorParameter;
	SetPositionProfile: FB_SetPositionProfile;
	SetOperationMode: FB_SetOperationMode;
	MoveToPosition: FB_MoveToPosition;
	GetMovementState: FB_GetMovementState;
	SetDisableState: FB_SetDisableState;
	SetPositionMust: FB_SetPositionMust;
	POSITION: DINT;
END_VAR

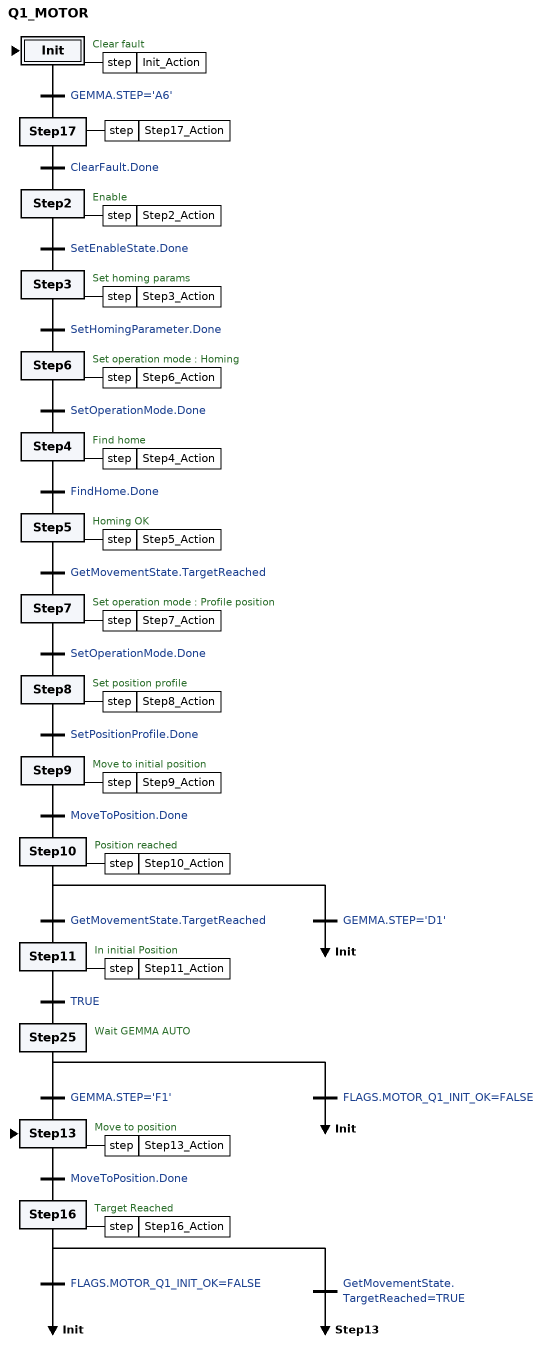
// Clear fault
INITIAL_STEP Init:
    Init_Action(N);  // step action
END_STEP
TRANSITION FROM Init TO Step17
    := GEMMA.STEP='A6';
END_TRANSITION
STEP Step17:
    Step17_Action(N);  // step action
END_STEP
TRANSITION FROM Step17 TO Step2
    := ClearFault.Done;
END_TRANSITION
// Enable
STEP Step2:
    Step2_Action(N);  // step action
END_STEP
TRANSITION FROM Step2 TO Step3
    := SetEnableState.Done;
END_TRANSITION
// Set homing params
STEP Step3:
    Step3_Action(N);  // step action
END_STEP
TRANSITION FROM Step3 TO Step6
    := SetHomingParameter.Done;
END_TRANSITION
// Set operation mode : Homing
STEP Step6:
    Step6_Action(N);  // step action
END_STEP
TRANSITION FROM Step6 TO Step4
    := SetOperationMode.Done;
END_TRANSITION
// Find home
STEP Step4:
    Step4_Action(N);  // step action
END_STEP
TRANSITION FROM Step4 TO Step5
    := FindHome.Done;
END_TRANSITION
// Homing OK
STEP Step5:
    Step5_Action(N);  // step action
END_STEP
TRANSITION FROM Step5 TO Step7
    := GetMovementState.TargetReached;
END_TRANSITION
// Set operation mode : Profile position
STEP Step7:
    Step7_Action(N);  // step action
END_STEP
TRANSITION FROM Step7 TO Step8
    := SetOperationMode.Done;
END_TRANSITION
// Set position profile
STEP Step8:
    Step8_Action(N);  // step action
END_STEP
TRANSITION FROM Step8 TO Step9
    := SetPositionProfile.Done;
END_TRANSITION
// Move to initial position
STEP Step9:
    Step9_Action(N);  // step action
END_STEP
TRANSITION FROM Step9 TO Step10
    := MoveToPosition.Done;
END_TRANSITION
// Position reached
STEP Step10:
    Step10_Action(N);  // step action
END_STEP
TRANSITION FROM Step10 TO Step11
    := GetMovementState.TargetReached;
END_TRANSITION
TRANSITION FROM Step10 TO Init
    := GEMMA.STEP='D1';
END_TRANSITION
// In initial Position
STEP Step11:
    Step11_Action(N);  // step action
END_STEP
TRANSITION FROM Step11 TO Step25
    := TRUE;
END_TRANSITION
// Wait GEMMA AUTO
STEP Step25:
END_STEP
TRANSITION FROM Step25 TO Step13
    := GEMMA.STEP='F1';
END_TRANSITION
TRANSITION FROM Step25 TO Init
    := FLAGS.MOTOR_Q1_INIT_OK=FALSE;
END_TRANSITION
// Move to position
STEP Step13:
    Step13_Action(N);  // step action
END_STEP
TRANSITION FROM Step13 TO Step16
    := MoveToPosition.Done;
END_TRANSITION
// Target Reached
STEP Step16:
    Step16_Action(N);  // step action
END_STEP
TRANSITION FROM Step16 TO Init
    := FLAGS.MOTOR_Q1_INIT_OK=FALSE;
END_TRANSITION
TRANSITION FROM Step16 TO Step13
    := GetMovementState.TargetReached=TRUE;
END_TRANSITION

ACTION Step10_Action:
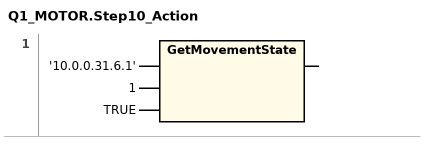
// NETWORK 1
GetMovementState('10.0.0.31.6.1', 1, TRUE);
END_ACTION

ACTION Step17_Action:
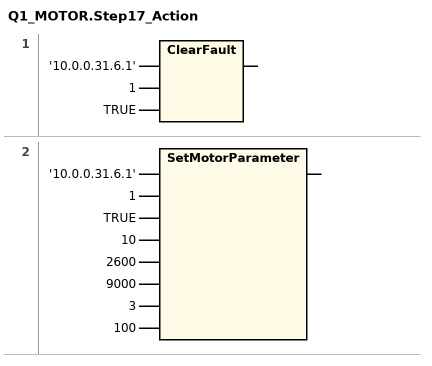
// NETWORK 1
ClearFault('10.0.0.31.6.1', 1, TRUE);

// NETWORK 2
SetMotorParameter('10.0.0.31.6.1', 1, TRUE, 10, 2600, 9000, 3, 100);
END_ACTION

ACTION Step13_Action:
(*Limitation deplacement Moteur*)
IF FLAGS.MOTOR_Q1_POSITION>MOTOR_Q1_POSITION_MAX THEN
	POSITION:=MOTOR_Q1_POSITION_MAX;
ELSIF FLAGS.MOTOR_Q1_POSITION<0 THEN
	POSITION:=0;
ELSE
	POSITION:=FLAGS.MOTOR_Q1_POSITION;
END_IF


MoveToPosition(
	ADSNetId:= '10.0.0.31.6.1',
	NodeId:= 1,
	Write:= TRUE,
	TargetPosition:= POSITION,
	Absolut:= TRUE);
END_ACTION

ACTION Step8_Action:
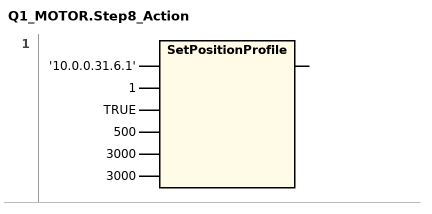
// NETWORK 1
SetPositionProfile('10.0.0.31.6.1', 1, TRUE, 500, 3000, 3000);
END_ACTION

ACTION Step16_Action:
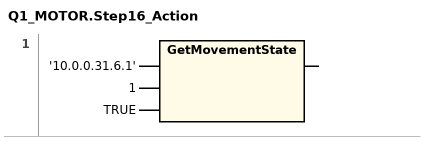
// NETWORK 1
GetMovementState('10.0.0.31.6.1', 1, TRUE);
END_ACTION

ACTION Step4_Action:
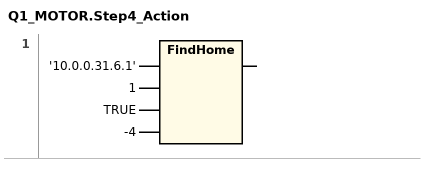
// NETWORK 1
FindHome('10.0.0.31.6.1', 1, TRUE, -4);
END_ACTION

ACTION Step3_Action:
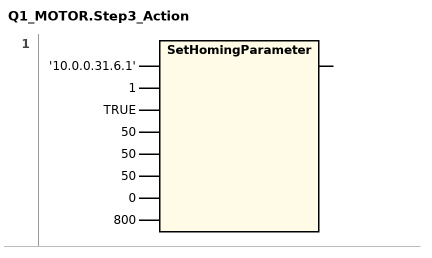
// NETWORK 1
SetHomingParameter('10.0.0.31.6.1', 1, TRUE, 50, 50, 50, 0, 800);
END_ACTION

ACTION Step5_Action:
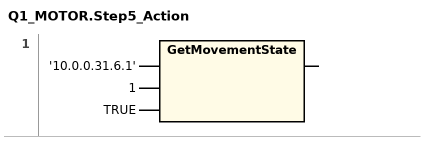
// NETWORK 1
GetMovementState('10.0.0.31.6.1', 1, TRUE);
END_ACTION

ACTION Step2_Action:
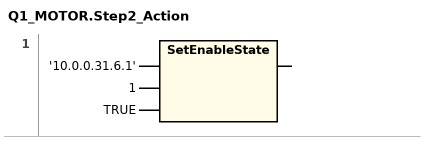
// NETWORK 1
SetEnableState('10.0.0.31.6.1', 1, TRUE);
END_ACTION

ACTION Init_Action:

END_ACTION

ACTION Step6_Action:
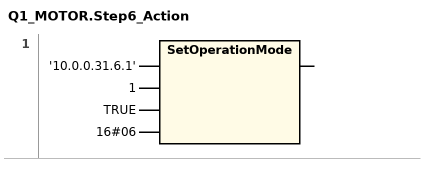
// NETWORK 1
SetOperationMode('10.0.0.31.6.1', 1, TRUE, 16#06);
END_ACTION

ACTION Step11_Action:

(*SetDisableState(
	ADSNetId:= '10.0.0.31.6.1',
	NodeId:= 1,
	Write:= TRUE);*)

FLAGS.MOTOR_Q1_INIT_OK:=TRUE;
END_ACTION

ACTION Step7_Action:
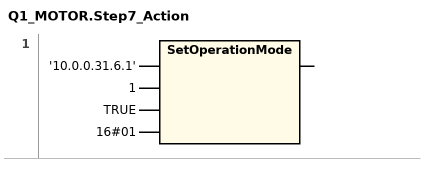
// NETWORK 1
SetOperationMode('10.0.0.31.6.1', 1, TRUE, 16#01);
END_ACTION

ACTION Step9_Action:
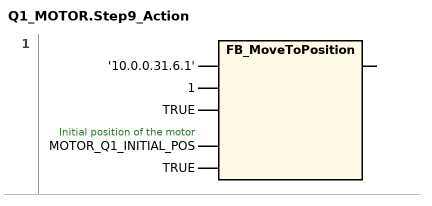
// NETWORK 1
//   MOTOR_Q1_INITIAL_POS: Initial position of the motor
FB_MoveToPosition('10.0.0.31.6.1', 1, TRUE, MOTOR_Q1_INITIAL_POS, TRUE);
END_ACTION

END_PROGRAM

// ---- POUs/Q2_MOTOR.TcPOU
PROGRAM Q2_MOTOR
VAR
	ClearFault: FB_ClearFault;
	SetEnableState: FB_SetEnableState;
	SetHomingParameter: FB_SetHomingParameter;
	FindHome: FB_FindHome;
	SetMotorParameter: FB_SetMotorParameter;
	SetPositionProfile: FB_SetPositionProfile;
	SetOperationMode: FB_SetOperationMode;
	MoveToPosition: FB_MoveToPosition;
	GetMovementState: FB_GetMovementState;
	SetDisableState: FB_SetDisableState;
	SetPositionMust: FB_SetPositionMust;
	POSITION: DINT;
END_VAR

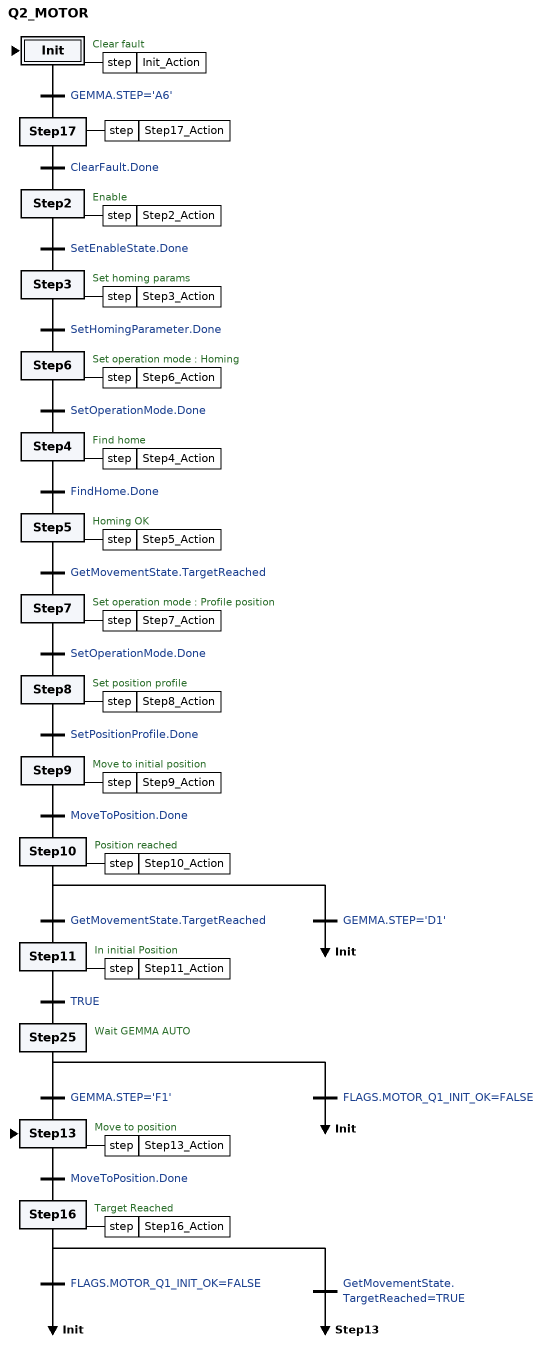
// Clear fault
INITIAL_STEP Init:
    Init_Action(N);  // step action
END_STEP
TRANSITION FROM Init TO Step17
    := GEMMA.STEP='A6';
END_TRANSITION
STEP Step17:
    Step17_Action(N);  // step action
END_STEP
TRANSITION FROM Step17 TO Step2
    := ClearFault.Done;
END_TRANSITION
// Enable
STEP Step2:
    Step2_Action(N);  // step action
END_STEP
TRANSITION FROM Step2 TO Step3
    := SetEnableState.Done;
END_TRANSITION
// Set homing params
STEP Step3:
    Step3_Action(N);  // step action
END_STEP
TRANSITION FROM Step3 TO Step6
    := SetHomingParameter.Done;
END_TRANSITION
// Set operation mode : Homing
STEP Step6:
    Step6_Action(N);  // step action
END_STEP
TRANSITION FROM Step6 TO Step4
    := SetOperationMode.Done;
END_TRANSITION
// Find home
STEP Step4:
    Step4_Action(N);  // step action
END_STEP
TRANSITION FROM Step4 TO Step5
    := FindHome.Done;
END_TRANSITION
// Homing OK
STEP Step5:
    Step5_Action(N);  // step action
END_STEP
TRANSITION FROM Step5 TO Step7
    := GetMovementState.TargetReached;
END_TRANSITION
// Set operation mode : Profile position
STEP Step7:
    Step7_Action(N);  // step action
END_STEP
TRANSITION FROM Step7 TO Step8
    := SetOperationMode.Done;
END_TRANSITION
// Set position profile
STEP Step8:
    Step8_Action(N);  // step action
END_STEP
TRANSITION FROM Step8 TO Step9
    := SetPositionProfile.Done;
END_TRANSITION
// Move to initial position
STEP Step9:
    Step9_Action(N);  // step action
END_STEP
TRANSITION FROM Step9 TO Step10
    := MoveToPosition.Done;
END_TRANSITION
// Position reached
STEP Step10:
    Step10_Action(N);  // step action
END_STEP
TRANSITION FROM Step10 TO Step11
    := GetMovementState.TargetReached;
END_TRANSITION
TRANSITION FROM Step10 TO Init
    := GEMMA.STEP='D1';
END_TRANSITION
// In initial Position
STEP Step11:
    Step11_Action(N);  // step action
END_STEP
TRANSITION FROM Step11 TO Step25
    := TRUE;
END_TRANSITION
// Wait GEMMA AUTO
STEP Step25:
END_STEP
TRANSITION FROM Step25 TO Step13
    := GEMMA.STEP='F1';
END_TRANSITION
TRANSITION FROM Step25 TO Init
    := FLAGS.MOTOR_Q1_INIT_OK=FALSE;
END_TRANSITION
// Move to position
STEP Step13:
    Step13_Action(N);  // step action
END_STEP
TRANSITION FROM Step13 TO Step16
    := MoveToPosition.Done;
END_TRANSITION
// Target Reached
STEP Step16:
    Step16_Action(N);  // step action
END_STEP
TRANSITION FROM Step16 TO Init
    := FLAGS.MOTOR_Q1_INIT_OK=FALSE;
END_TRANSITION
TRANSITION FROM Step16 TO Step13
    := GetMovementState.TargetReached=TRUE;
END_TRANSITION

ACTION Step17_Action:
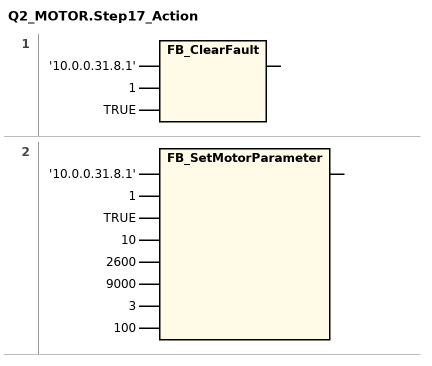
// NETWORK 1
FB_ClearFault('10.0.0.31.8.1', 1, TRUE);

// NETWORK 2
FB_SetMotorParameter('10.0.0.31.8.1', 1, TRUE, 10, 2600, 9000, 3, 100);
END_ACTION

ACTION Step4_Action:
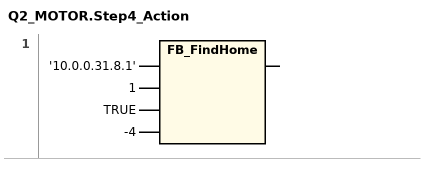
// NETWORK 1
FB_FindHome('10.0.0.31.8.1', 1, TRUE, -4);
END_ACTION

ACTION Step2_Action:
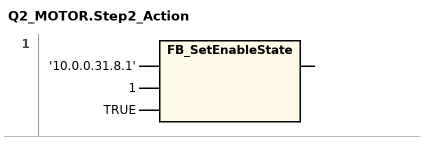
// NETWORK 1
FB_SetEnableState('10.0.0.31.8.1', 1, TRUE);
END_ACTION

ACTION Step13_Action:
(*Limitation deplacement Moteur*)
IF FLAGS.MOTOR_Q2_POSITION>MOTOR_Q2_POSITION_MAX THEN
	POSITION:=MOTOR_Q2_POSITION_MAX;
ELSIF FLAGS.MOTOR_Q2_POSITION<0 THEN
	POSITION:=0;
ELSE
	POSITION:=FLAGS.MOTOR_Q2_POSITION;
END_IF


MoveToPosition(
	ADSNetId:= '10.0.0.31.8.1',
	NodeId:= 1,
	Write:= TRUE,
	TargetPosition:= POSITION,
	Absolut:= TRUE);
END_ACTION

ACTION Step10_Action:
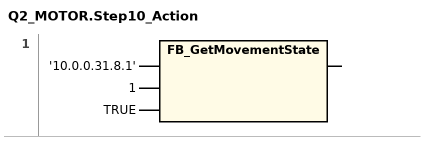
// NETWORK 1
FB_GetMovementState('10.0.0.31.8.1', 1, TRUE);
END_ACTION

ACTION Step5_Action:
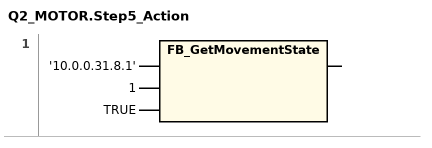
// NETWORK 1
FB_GetMovementState('10.0.0.31.8.1', 1, TRUE);
END_ACTION

ACTION Step7_Action:
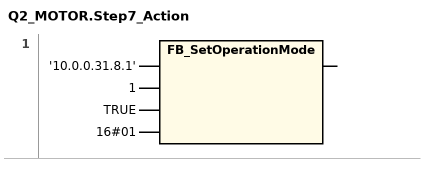
// NETWORK 1
FB_SetOperationMode('10.0.0.31.8.1', 1, TRUE, 16#01);
END_ACTION

ACTION Step9_Action:
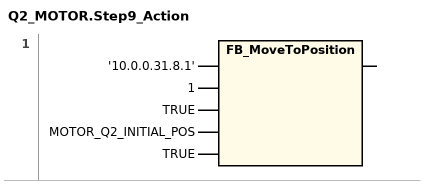
// NETWORK 1
FB_MoveToPosition('10.0.0.31.8.1', 1, TRUE, MOTOR_Q2_INITIAL_POS, TRUE);
END_ACTION

ACTION Step11_Action:

(*SetDisableState(
	ADSNetId:= '10.0.0.31.6.1',
	NodeId:= 1,
	Write:= TRUE);*)

FLAGS.MOTOR_Q2_INIT_OK:=TRUE;
END_ACTION

ACTION Step3_Action:
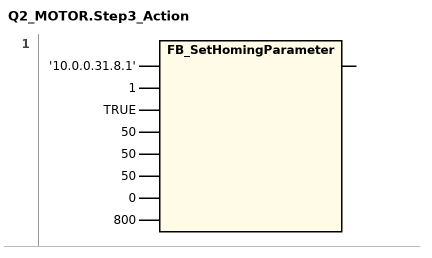
// NETWORK 1
FB_SetHomingParameter('10.0.0.31.8.1', 1, TRUE, 50, 50, 50, 0, 800);
END_ACTION

ACTION Step6_Action:
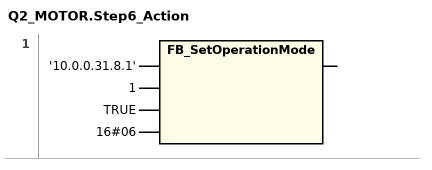
// NETWORK 1
FB_SetOperationMode('10.0.0.31.8.1', 1, TRUE, 16#06);
END_ACTION

ACTION Init_Action:

END_ACTION

ACTION Step16_Action:
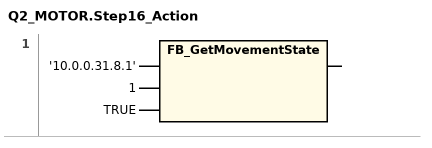
// NETWORK 1
FB_GetMovementState('10.0.0.31.8.1', 1, TRUE);
END_ACTION

ACTION Step8_Action:
